	MP_BAK							: sMachPara;
END_VAR
VAR_IN_OUT
	sVisu : sMPHandler;
END_VAR
DisableMP();
j:=1;
FOR i:=1 TO 20 DO
	IF ExportDirectory[i].sFileName<>''
	THEN
		sVisu.FileListExport[j]:=ExportDirectory[i].sFileName;
		j:=j+1;
	ELSE
		sVisu.FileListExport[j]:='';
		j:=j+1;
	END_IF
END_FOR
j:=1;
FOR i:=1 TO 20 DO
	IF LocalDirectory[i].sFileName<>''
	THEN
		sVisu.FileListLocal[j]:=LocalDirectory[i].sFileName;
		j:=j+1;
	ELSE
		sVisu.FileListLocal[j]:='';
		j:=j+1;
	END_IF
END_FOR


(* --------------------------------------------------------------- *)
(* -----------------  sVisu interface ----------------------------- *)
(* --------------------------------------------------------------- *)



BtnImport(
	Enable			:= StepExport=0,
	Visible			:= FALSE,
	TextOn			:= 'Import',
	TextOff			:= 'Import',
	Button			:= sVisu.BtnImport
  );



BtnExport(
	Enable			:= StepExport=0,
	Visible			:= TRUE,
	TextOn			:= 'Export',
	TextOff			:= 'Export',
	Button			:= sVisu.BtnExport
  );

IF BtnExport.PressedFlag
THEN
StepExport:=1;

END_IF


CASE StepExport OF
(* Überprüfen ob Laufwerk vorh. ist *)
	0:	sVisu.MessageString:='';
	1:	FileNameSearchExport	:=	MP_ExportDrive;
			sVisu.MessageString:='';
			StepExport			:=	2(*2*);
	2:	FileListUpdateExport:=TRUE;
			StepExport			:=	3;
	3:	IF ExportFiles.bError OR (ExportFiles.bEOE AND ExportFiles.nFindFiles=0 AND NOT ExportFiles.bBusy)
			THEN
				sVisu.MessageString:='Exportlaufwerk wurde nichterkannt!';
				FileListUpdateExport:=FALSE;
				StepExport			:=	999;
			ELSIF ExportFiles.bEOE AND  ExportFiles.nFindFiles>0
			THEN
				FileListUpdateExport:=FALSE;
				StepExport			:=	4;
			END_IF
	4:	IF NOT ExportFiles.bBusy
			THEN
				StepExport			:=	10;
			END_IF
(* Typdaten Exportpfad prüfen / anlegen *)
	10:	FileNameSearchExport	:=	MP_ExportDrivePathTD;(* 4 *)
			sVisu.MessageString:='';
			StepExport			:=	11;
	11:	FileListUpdateExport:=TRUE;
			StepExport			:=	12;
	12:	IF ExportFiles.nFindFiles=0 AND (ExportFiles.bEOE OR ExportFiles.bError)
			THEN
				sVisu.MessageString:='Typdatenpfad wird angelegt! -> /_TD/';
				FileListUpdateExport:=FALSE;
				StepExport			:=	13;
			ELSIF ExportFiles.nFindFiles>0 AND (ExportFiles.bEOE OR ExportFiles.bError)
			THEN
				FileListUpdateExport:=FALSE;
				StepExport			:=	20;
			END_IF
	13:	CreateDirectory.sPathName:=MP_ExportDrivePathTD;
			CreateDirectory.bExecute:=FALSE;
			StepExport			:=	14;
	14:	CreateDirectory.bExecute:=TRUE;
			IF CreateDirectory.bBusy
			THEN
				StepExport			:=	15;
			END_IF
	15:	IF NOT CreateDirectory.bBusy AND NOT CreateDirectory.bError
			THEN
				StepExport			:=	20;

			ELSIF NOT CreateDirectory.bBusy AND CreateDirectory.bError
			THEN
				StepExport			:=	999;
				sVisu.MessageString:='Fehler bein erstellen des Typdatenpfades';
			END_IF


(* Maschinenparameter Exportpfad prüfen / anlegen *)
	20:	FileNameSearchExport	:=	MP_ExportDrivePathMP;
			sVisu.MessageString:='';
			StepExport			:=	21;
	21:	FileListUpdateExport:=TRUE;
			StepExport			:=	22;
	22:	IF ExportFiles.nFindFiles=0 AND (ExportFiles.bEOE OR ExportFiles.bError)
			THEN
				sVisu.MessageString:='Maschinenparameterpfad  wird angelegt! -> /_MP/';
				FileListUpdateExport:=FALSE;
				StepExport			:=	23;
			ELSIF ExportFiles.nFindFiles>0 AND (ExportFiles.bEOE OR ExportFiles.bError)
			THEN
				FileListUpdateExport:=FALSE;
				StepExport			:=	40;
			END_IF
	23:	CreateDirectory.sPathName:=MP_ExportDrivePathMP;
			CreateDirectory.bExecute:=FALSE;
			StepExport			:=	24;
	24:	CreateDirectory.bExecute:=TRUE;
			IF CreateDirectory.bBusy
			THEN
				StepExport			:=	25;
			END_IF
	25:	IF NOT CreateDirectory.bBusy AND NOT CreateDirectory.bError
			THEN
				StepExport			:=	40;

			ELSIF NOT CreateDirectory.bBusy AND CreateDirectory.bError
			THEN
				StepExport			:=	999;
				sVisu.MessageString:='Fehler bein erstellen des Maschinenparameterpfades';
			END_IF

	(* Typdaten kopieren *)
	40: sVisu.MessageString:='';
			StepExport			:=	41;
			FileNameSearchExport	:=	CONCAT(CONCAT(MP_ExportDrivePathTD,Backslash),MP_TDSearchString);
			FileNameSearchLocal		:=	CONCAT(MP_TDPathLocal,MP_TDSearchString);
	41: FileListUpdateExport:=TRUE;
			StepExport			:=	42;
	42: IF ExportFiles.bEOE OR ExportFiles.bError
			THEN
				FileListUpdateExport:=FALSE;
				StepExport			:=	43;
			END_IF
	43: FileListUpdateLocal:=TRUE;
			StepExport			:=	44;
	44: IF LocalFiles.nFindFiles=0 AND (LocalFiles.bEOE OR LocalFiles.bError)
			THEN
				sVisu.MessageString:='Es wurden keine Typdaten zum Exportieren gefunden!';
				FileListUpdateLocal:=FALSE;
				StepExport			:=	100;
			ELSIF LocalFiles.nFindFiles>0 AND (LocalFiles.bEOE OR LocalFiles.bError)
			THEN
				FileListUpdateLocal:=FALSE;
				NoOfTDFilesToCopy:=LocalFiles.nFindFiles;
				StepExport			:=	60;
			END_IF

	60:	AktFileToCopy		:=	1;
			StepExport			:=	61;

	61: (* Set Path *)
			TempStringSource					:=	CONCAT(MP_TDPathLocal,LocalDirectory[AktFileToCopy].sFileName);
			TempStringTarget					:=	CONCAT(CONCAT(MP_ExportDrivePathTD,Backslash),LocalDirectory[AktFileToCopy].sFileName);
			CopyFiles.srcFileName			:=	TempStringSource;
			CopyFiles.destFileName		:=	TempStringTarget;
			CopyFiles.bExecute				:=	FALSE;
			StepExport								:=	62;
			sVisu.MessageString:='Typdaten werden kopiert...';

	62: (* Start to Copy *)
			CopyFiles.bExecute				:=	TRUE;
			IF CopyFiles.bBusy
			THEN
				StepExport								:=	63;
			END_IF
	63: (* Copy Done *)
			CopyFiles.bExecute				:=	FALSE;
			IF NOT CopyFiles.bBusy AND NOT CopyFiles.bError
			THEN
				StepExport								:=	64;
			ELSIF NOT CopyFiles.bBusy AND CopyFiles.bError
			THEN
				StepExport								:=	999;
				sVisu.MessageString:='Fehler beim kopieren der Typdaten!';
			END_IF
	64: FileListUpdateExport:=TRUE;
			StepExport			:=	65;
	65:	(* Check last file To copy *)
			FileListUpdateExport:=FALSE;
			IF AktFileToCopy>=NoOfTDFilesToCopy
			THEN
				StepExport								:=	66;
			ELSE
				AktFileToCopy							:=	AktFileToCopy + 1;
				StepExport								:=	61;
			END_IF

	66:	(* All Files copied *)
			sVisu.MessageString:='Typdaten kopieren abgeschlossen!';
				StepExport								:=	100;

 100:	(* Maschinendaten sichern *)
			WriteXML.bExecute					:=	FALSE;
			StepExport								:=	101;
 101: WriteXML.bExecute					:=	TRUE;
			IF WriteXML.bBusy
			THEN
				WriteXML.bExecute					:=	FALSE;
				StepExport								:=	102;
			END_IF
 102: IF NOT WriteXML.bBusy AND NOT WriteXML.bError
			THEN
				WriteXML.bExecute					:=	FALSE;
				StepExport								:=	110;
			ELSIF NOT WriteXML.bBusy AND WriteXML.bError
			THEN
				sVisu.MessageString:='Fehler bein schreiben der XML-Datei für die Maschinenparameter....';
				WriteXML.bExecute					:=	FALSE;
				StepExport								:=	999;
			END_IF
 110:
			(* Set Path *)
			TempStringSource					:=	CONCAT(CONCAT(MP_ExportDrivePathMP, Backslash),MP_MPExportFilename);(*'\Hard Disk\_MP\MachPara.xml';*)
			TempStringTarget					:=	CONCAT(CONCAT(MP_ExportDrivePathMP, Backslash),MP_MPExportFilename);(*'\Hard Disk2\_MP\MachPara.xml';*)
			CopyFiles.srcFileName			:=	TempStringSource;
			CopyFiles.destFileName		:=	TempStringTarget;
			CopyFiles.bExecute				:=	FALSE;
			StepExport								:=	111;
			sVisu.MessageString:='Maschinenparameter werden kopiert...';

	111: (* Start to Copy *)
			CopyFiles.bExecute				:=	TRUE;
			IF CopyFiles.bBusy
			THEN
				StepExport								:=	112;
			END_IF
	112: (* Copy Done *)
			CopyFiles.bExecute				:=	FALSE;
			IF NOT CopyFiles.bBusy AND NOT CopyFiles.bError
			THEN
				sVisu.MessageString:='Maschinenparameter kopieren abgeschlossen!';
				StepExport								:=	999;
			ELSIF NOT CopyFiles.bBusy AND CopyFiles.bError
			THEN
				StepExport								:=	999;
				sVisu.MessageString:='Fehler beim kopieren der Maschinenparameter!';
			END_IF
 999:	Delay(IN:= FALSE, PT:= t#0s);
			StepExport			:=	1000;
1000: Delay(IN:= TRUE, PT:= t#1s);
			IF delay.Q
			THEN
				StepExport			:=	0;
			END_IF
END_CASE


ExportFiles(
	bExecute			:=sVisu.FileListUpdate OR FileListUpdateExport,
	sNetId				:= '',
	sPathName			:= FileNameSearchExport,
	pFindList			:= ADR(ExportDirectory),
	cbFindList		:= SIZEOF(ExportDirectory) ,
	tTimeout			:= t#10s );

LocalFiles(
	bExecute			:=sVisu.FileListUpdate OR FileListUpdateLocal,
	sNetId				:= '',
	sPathName			:= FileNameSearchLocal,
	pFindList			:= ADR(LocalDirectory),
	cbFindList		:= SIZEOF(LocalDirectory) ,
	tTimeout			:= t#1s );

CopyFiles(
	srcNetId:= '',
	destNetId:= '',
	tAdsSTATE_TIMEOUT:= t#1s);


WriteXML(
	sNetId				:= '',
	nMode					:= XMLSRV_ADDMISSING,
 	sSymName				:='.MP',
	sFilePath			:= CONCAT(CONCAT(MP_ExportDrivePathMP, Backslash),MP_MPExportFilename),
	sXPath				:= '/dataentry/MP',
	tTimeout			:= t#10s );


sVisu.FileListUpdate:=FALSE;

CreateDirectory(
	sNetId:= '' );


ReadXML(
	sNetId:= '',
	nMode:= XMLSRV_ADDMISSING,
	sSymName:= '.MP',
	sFilePath:= '\Hard Disk\_MP\MachPara.xml',
	sXPath:= '/dataentry/MP'
);


IF MEMCMP(ADR(MP),ADR(MP_BAK),SIZEOF(MP_BAK))<>0
THEN
	Visu.SavePersistentData:=TRUE;
	MP_BAK:=MP;
END_IF
END_PROGRAM
ACTION DisableMP:
(* Sperre der Typdateneingabe *)
gDisableMP := FALSE;
IF 	CurrentUserLevel <6  OR
	ModeSelect.Mode > MODE_MANUAL THEN
	gDisableMP := TRUE;
END_IF
END_ACTION

(* POU System/HelpFunctions/FB_FileCopy, ST *)
FUNCTION_BLOCK FB_FileCopy
VAR_INPUT
	srcNetId				: T_AmsNetId;	(* TwinCAT network address of the source file *)
	srcFileName				: T_MaxString;	(* source file path and name *)
	destNetId				: T_AmsNetId;	(* TwinCAT network address of the destination file *)
	destFileName			: T_MaxString;  	(* destination file path and name *)
	bExecute				: BOOL;		(* rising edge starts fb execution *)
	tAdsSTATE_TIMEOUT	: TIME;		(* ads STATE_TIMEOUT *)
END_VAR
VAR_OUTPUT
	bBusy		  		:BOOL;
	bError				:BOOL;
	nErrId				:UDINT;
END_VAR
VAR
	fbFileOpen			:FB_FileOpen;
	fbFileClose			:FB_FileClose;
	fbFileRead			:FB_FileRead;
	fbFileWrite			:FB_FileWrite;

	hSrcFile				:UINT	:= 0;(* file handle of the source file *)
	hDestFile			:UINT	:= 0;(* file handle of the destination file *)

	Step				:DWORD;
	RisingEdge			:R_TRIG;

	buffRead			:ARRAY[1..100000] OF BYTE;(* buffer *)
	cbReadLength		:UDINT:=0;
END_VAR
RisingEdge(CLK:=bExecute);
IF RisingEdge.Q THEN
	IF 	NOT bBusy THEN
		bBusy := TRUE;
		bError:= FALSE;
		nErrId:=0;
		Step := 1;
		cbReadLength:=0;
		hSrcFile:=0;
		hDestFile:=0;
	END_IF
END_IF


CASE Step OF
	0:(* do nothing *)
	;

	1:(* open source file *)
	fbFileOpen(  bExecute := FALSE  );
	fbFileOpen(	sNetId := srcNetId,
		sPathName := srcFileName,
		nMode := FOPEN_MODEREAD OR FOPEN_MODETEXT ,
		ePath := PATH_GENERIC,
		tTimeout := tAdsSTATE_TIMEOUT,
		bExecute := TRUE );
		Step := Step + 1;

	2:
	fbFileOpen( bExecute := FALSE );
	IF ( NOT fbFileOpen.bBusy ) THEN
		IF ( fbFileOpen.bError ) THEN
			nErrId := fbFileOpen.nErrId;
			bError := TRUE;
			Step := 50;
		ELSE
			hSrcFile := fbFileOpen.hFile;
			Step := Step + 1;
		END_IF
	END_IF

	3:(* open destination file *)
	fbFileOpen(  bExecute := FALSE  );
	fbFileOpen( 	sNetId := destNetId,
			sPathName := destFileName,
			nMode := FOPEN_MODEWRITE OR FOPEN_MODETEXT ,
			ePath := PATH_GENERIC,
			tTimeout := tAdsSTATE_TIMEOUT,
			bExecute := TRUE );
	Step := Step+1;

	4:
	fbFileOpen(  bExecute := FALSE  );
	IF ( NOT fbFileOpen.bBusy ) THEN
		IF ( fbFileOpen.bError ) THEN
			nErrId := fbFileOpen.nErrId;
			bError := TRUE;
			Step := 50;
		ELSE
			hDestFile := fbFileOpen.hFile;
			Step := Step + 1;
		END_IF
	END_IF

	5:(*read data from source file*)
	cbReadLength := 0;
	fbFileRead( bExecute:= FALSE );
	fbFileRead( 	sNetId:=SrcNetId,
			hFile:=hSrcFile,
			pReadBuff:= ADR(buffRead),
			cbReadLen:= SIZEOF(buffRead),
			bExecute:=TRUE,
			tTimeout:=tAdsSTATE_TIMEOUT );
	Step := Step + 1;

	6:
	fbFileRead( bExecute:= FALSE );
	IF ( NOT fbFileRead.bBusy ) THEN
		IF ( fbFileRead.bError ) THEN
			nErrId := fbFileRead.nErrId;
			bError := TRUE;
			Step := 50;
		ELSE
			cbReadLength := fbFileRead.cbRead;
			Step := Step + 1;
		END_IF
	END_IF

	7:(*write data to destination file*)
	fbFileWrite( bExecute := FALSE );
	fbFileWrite(	sNetId:=DestNetId,
			hFile:=hDestFile,
			pWriteBuff:= ADR(buffRead),
			cbWriteLen:= cbReadLength,
			bExecute:=TRUE,
			tTimeout:=tAdsSTATE_TIMEOUT );
	Step := Step + 1;

	8:
	fbFileWrite( bExecute := FALSE );
	IF ( NOT fbFileWrite.bBusy ) THEN
		IF ( fbFileWrite.bError ) THEN
			nErrId := fbFileWrite.nErrId;
			bError := TRUE;
			Step := 50;
		ELSE
			IF fbFileRead.bEOF THEN (*Check if the EOF flag ist set *)
				Step := 50;(*cleanup: close the destination and source files *)
			ELSE
				Step := 5; (* repeat reading *)
			END_IF
		END_IF
	END_IF

	30:(* close the destination file *)
	fbFileClose( bExecute := FALSE );
	fbFileClose( 	sNetId:=destNetId,
			hFile:=hDestFile,
			bExecute:=TRUE,
			tTimeout:=tAdsSTATE_TIMEOUT );
	Step := Step + 1;

	31:
	fbFileClose( bExecute := FALSE );
	IF ( NOT fbFileClose.bBusy ) THEN
		IF ( fbFileClose.bError ) THEN
			nErrId := fbFileClose.nErrId;
			bError := TRUE;
		END_IF
		Step := 50;
		hDestFile := 0;
	END_IF

	40: (* close source file *)
	fbFileClose( bExecute := FALSE );
	fbFileClose( 	sNetId:=srcNetId,
			hFile:=hSrcFile,
			bExecute:=TRUE,
			tTimeout:=tAdsSTATE_TIMEOUT );
	Step := Step + 1;

	41:
	fbFileClose( bExecute := FALSE );
	IF ( NOT fbFileClose.bBusy ) THEN
		IF ( fbFileClose.bError ) THEN
			nErrId := fbFileClose.nErrId;
			bError := TRUE;
		END_IF
		Step := 50;
		hSrcFile := 0;
	END_IF

	50: (*error or ready => cleanup*)
	IF ( hDestFile <> 0 ) THEN
		Step := 30; (* close the destination file*)
	ELSIF (hSrcFile <> 0 ) THEN
		Step := 40; (* close the source file *)
	ELSE
		Step := 0;	(* ready *)
		bBusy := FALSE;
	END_IF

END_CASE
END_FUNCTION_BLOCK

(* POU System/MP_ShiftHandler/MP_ShiftHandler, ST *)
PROGRAM MP_ShiftHandler
VAR
	TodNow				: TOD;

	TempStartTOD 		: TOD;
	TempEndTOD 			: TOD;

	TempNightShift		: BOOL;

	TimeDayBegins		: TOD := TOD#00:00;
	TimeDayEnds			: TOD := TOD#23:59:59.999;

	NumberofShifts		: DINT;
	Idx					: DINT;

	NoShiftActive		: sMP_ShiftData;
	OneShiftIsActive	: BOOL;

END_VAR
NoShiftActive.ShiftIndex:=999;
NoShiftActive.ShiftName:='keine Schicht Activ';


NumberofShifts:=SIZEOF(MP.ShiftData.Shift)/SIZEOF(mp.ShiftData.ActiveShift);

TodNow:=DT_TO_TOD(SYSTEMTIME_TO_DT(gVarSystemtime));
TodNow:=	DINT_TO_TOD(TOD_TO_DINT(TodNow)	+	WORD_TO_DINT(gVarSystemtime.wMilliseconds));


OneShiftIsActive:=FALSE;

FOR Idx:=1 TO NumberofShifts DO


	MP.ShiftData.Shift[Idx].TimeStart.wYear:=gVarSystemtime.wYear;
	MP.ShiftData.Shift[Idx].TimeStart.wMonth:=gVarSystemtime.wMonth;
	MP.ShiftData.Shift[Idx].TimeStart.wDay:=gVarSystemtime.wDay;
	MP.ShiftData.Shift[Idx].TimeStart.wDayOfWeek:=gVarSystemtime.wDayOfWeek;
	MP.ShiftData.Shift[Idx].TimeStart.wSecond:=0;
	MP.ShiftData.Shift[Idx].TimeStart.wMilliseconds:=0;


	MP.ShiftData.Shift[Idx].TimeEnd.wYear:=gVarSystemtime.wYear;
	MP.ShiftData.Shift[Idx].TimeEnd.wMonth:=gVarSystemtime.wMonth;
	MP.ShiftData.Shift[Idx].TimeEnd.wDay:=gVarSystemtime.wDay;
	MP.ShiftData.Shift[Idx].TimeEnd.wDayOfWeek:=gVarSystemtime.wDayOfWeek;
	MP.ShiftData.Shift[Idx].TimeEnd.wSecond:=59;
	MP.ShiftData.Shift[Idx].TimeEnd.wMilliseconds:=0;


	TempStartTOD:=DT_TO_TOD(SYSTEMTIME_TO_DT(MP.ShiftData.Shift[Idx].TimeStart));

	TempStartTOD:=	DINT_TO_TOD(TOD_TO_DINT(TempStartTOD)	+	WORD_TO_DINT(MP.ShiftData.Shift[Idx].TimeStart.wMilliseconds));

	TempEndTOD:=DT_TO_TOD(SYSTEMTIME_TO_DT(MP.ShiftData.Shift[Idx].TimeEnd));

	MP.ShiftData.Shift[Idx].TimeEnd.wMilliseconds:=999;
	TempEndTOD:=	DINT_TO_TOD(TOD_TO_DINT(TempEndTOD)	+	WORD_TO_DINT(MP.ShiftData.Shift[Idx].TimeEnd.wMilliseconds));


	TempNightShift:=TOD_TO_DINT(TempStartTOD)>TOD_TO_DINT(TempEndTOD);

	IF 	NOT TempNightShift THEN
		MP.ShiftData.Shift[Idx].ShiftActive:=	(TodNow >= TempStartTOD)	AND (TodNow <= TempEndTOD);
	ELSE
		MP.ShiftData.Shift[Idx].ShiftActive:=	(TodNow >= TempStartTOD) AND
											(TodNow <= TimeDayEnds) OR (TodNow >= TimeDayBegins) AND
											(TodNow <= TempEndTOD);
	END_IF

	IF 	NOT OneShiftIsActive THEN
		OneShiftIsActive:=MP.ShiftData.Shift[Idx].ShiftActive;
		MP.ShiftData.ActiveShift:=MP.ShiftData.Shift[Idx];
	END_IF

END_FOR

IF 	NOT OneShiftIsActive THEN
	MP.ShiftData.ActiveShift:=NoShiftActive;
END_IF
END_PROGRAM

(* POU Stations/ST_00/ST00_FBs/_CallFBs, ST *)
PROGRAM _CallFBs


VAR



END_VAR
ST00_CallFBs();
ST03_CallFBs();

ST08_CallFBs();
END_PROGRAM

(* POU Stations/ST_00/ST00_FBs/ST00_CallFBs, ST *)
PROGRAM ST00_CallFBs
(*   Author:           *)


VAR



END_VAR
(* ----------------------------------------------------------------------------------------- *)
(* 																				Eingänge  																				 *)
(* ----------------------------------------------------------------------------------------- *)


(* Call ST00_40_F1 Vorsicherungen Leistung iO (DigIn) *)
ST00_40_F1(	sVisu:=Visu.ST00_40_F1,
			Reset:=gResetAll,
			CheckSignalHigh:=TRUE,
);

(* Call ST03_210_S1 Not-Aus 1 Anlage ausgelöst (DigIn) *)
ST03_210_S1(	sVisu:=Visu.ST03_210_S1,
				Reset:=gResetAll,
				CheckSignalLow:=TRUE,
);
(* Call ST08_210_S2 Not-Aus 2 Anlage ausgelöst (DigIn) *)
ST08_210_S2(	sVisu:=Visu.ST08_210_S2,
				Reset:=gResetAll,
				CheckSignalLow:=FALSE,
				CheckSignalHigh:=TRUE,
);

(* Call ST00_X4_16  Not-Halt 2 Tampondrucker  (DigIn) *)
ST00_X4_16(	sVisu:=Visu.ST00_X4_16,
			Reset:=gResetAll,
			CheckSignalLow:=TRUE,
);

(* Call ST00_200_A1_A1 Not-Aus iO (DigIn) *)
ST00_200_A1_A1(	sVisu:=Visu.ST00_200_A1_A1,
				Reset:=gResetAll,
				CheckSignalHigh:=TRUE,
);

(* Call ST00_220_S1 Schutztüre 1 geöffnet (DigIn) *)
ST00_220_S1(sVisu:=Visu.ST00_220_S1,
			Reset:=gResetAll,
			CheckSignalLow:=TRUE,
);

(* Call ST00_220_S2 Schutztüre 1 geöffnet (DigIn) *)
ST00_220_S2(sVisu:=Visu.ST00_220_S2,
			Reset:=gResetAll,
			CheckSignalLow:=TRUE,
);

(* Call ST00_230_S2_E1 Schutztüre 1 geschlossen (DigIn) *)
ST00_230_S2_E1(sVisu:=Visu.ST00_230_S2_E1,
			Reset:=gResetAll,
			(* CheckSignalHigh:=TRUE,*) (* @@@ *)
);

(* Call ST00_240_S1 Schutztüre 9 geschlossen (DigIn) *)
ST00_240_S1(sVisu:=Visu.ST00_240_S1,
			Reset:=gResetAll,
);

(* Call ST00_226_S1 Hubtüre 1 Schleuse Einlauf STN 8 geschlossen (DigIn) *)
ST00_226_S1(sVisu:=Visu.ST00_226_S1,
			Reset:=gResetAll,
);
(* Call ST00_226_S2 Hubtüre 2 Schleuse Einlauf STN 8 geschlossen (DigIn) *)
ST00_226_S2(sVisu:=Visu.ST00_226_S2,
			Reset:=gResetAll,
);
(* Call ST00_227_S1 Hubtüre 3 Schleuse Auslauf STN 8 geschlossen (DigIn) *)
ST00_227_S1(sVisu:=Visu.ST00_227_S1,
			Reset:=gResetAll,
);
(* Call ST00_227_S2 Hubtüre 4 Schleuse Auslauf STN 8 geschlossen (DigIn) *)
ST00_227_S2(sVisu:=Visu.ST00_227_S2,
			Reset:=gResetAll,
);
(* Call ST00_229_S1 Schutztüre Einlauf Tray STN 8 geschlossen (DigIn) *)
ST00_229_S1(sVisu:=Visu.ST00_229_S1,
			Reset:=gResetAll,
);
(* Call ST00_230_S1 Schutztüre Auslauf Tray STN 8 geschlossen (DigIn) *)
ST00_230_S1(sVisu:=Visu.ST00_230_S1,
			Reset:=gResetAll,
);
(* Call ST00_231_S1 Schutztüre Panel / Rutsche STN 8 geschlossen (DigIn) *)
ST00_231_S1(sVisu:=Visu.ST00_231_S1,
			Reset:=gResetAll,
);
(* Call ST00_232_S1 Schutztüre 8 Auslauf Tray STN 8 geschlossen (DigIn) *)
ST00_232_S1(sVisu:=Visu.ST00_232_S1,
			Reset:=gResetAll,
);
(* Call ST00_170Motorschutz Motorschutz in Ordnung (DigIn) *)
ST00_170_Motorschutz( sVisu:=Visu.ST00_170_Motorschutz,
						Reset:=gResetAll,
						CheckSignalHigh:=TRUE,
);

(* Call ST00_Thermokont Thermokontakt in Ordnung (DigIn) *)
ST00_170_Thermokont(	sVisu:=Visu.ST00_170_Thermokont,
						Reset:=gResetAll,
						CheckSignalHigh:=TRUE,
);


(* Call ST00_228_S1 Pallettierer in Position (DigIn) *)
ST00_228_S1(sVisu:=Visu.ST00_228_S1,
			Reset:=gResetAll,
);

(* Call ST00_71_X1_3 Schnittstelle Bedrucken Tinte JSK auf Übergabeposition (DigIn) *)
ST00_71_X1_3(sVisu:=Visu.ST00_71_X1_3,
			Reset:=gResetAll,
);

(* Call ST00_71_X1_4 Schnittstelle Bedrucken Tinte Druckstation betriebsbereit (DigIn) *)
ST00_71_X1_4(sVisu:=Visu.ST00_71_X1_4,
			Reset:=gResetAll,
);

(* Call ST00_72_X1_3 Schnittstelle Tampondrucker Teil in Abholposition (DigIn) *)(*Band Entnahmeposition 1*)
ST00_72_X1_3(sVisu:=Visu.ST00_72_X1_3,
			Reset:=gResetAll,
);

(* Call ST00_72_X1_8 Schnittstelle Tampondrucker Druck abgeschlossen (DigIn) *)
ST00_72_X1_8(sVisu:=Visu.ST00_72_X1_8,
			Reset:=gResetAll,
);

(* Call ST00_292_S1_STOP Bedienstelle Produktion Stop (DigIn) *)
ST00_292_S1_STOP(	sVisu:=Visu.ST00_292_S1_STOP,
					Reset:=gResetAll,
);
(* Call ST00_292_S2_START Bedienstelle Produktion Start (DigIn) *)
ST00_292_S2_START(	sVisu:=Visu.ST00_292_S2_START,
					Reset:=gResetAll,
);

(* Call ST00_292_S3_RESET Bedienstelle Produktion Start (DigIn) *)
ST00_292_S3_RESET(	sVisu:=Visu.ST00_292_S3_RESET,
					Reset:=gResetAll,
);
(* Call ST00_350_B20_0 Druckschalter Wartungseinheit Hauptluft min.6 bar (DigIn) *)
ST00_350_B20_0(	sVisu:=Visu.ST00_350_B20_0,
				Reset:=gResetAll,
				CheckSignalHigh:=TRUE,
);

(* Call 	ST00_245_V1			Verriegelung Schutztüren-Leuchte (DigOutIn) *)
ST00_245_V1(	sVisu:=Visu.ST00_245_V1,
					Reset:=gResetAll,
);

(* Call 	ST00_245_V2_START	Bedienstelle Start-Leuchte (DigOutIn) *)
ST00_245_V2_START(	sVisu:=Visu.ST00_245_V2_START,
					Reset:=gResetAll,
);

(* Call 	ST00_245_V3_RESET	Bedienstelle Reset-Schutztüren-Leuchte (DigOutIn) *)
ST00_245_V3_RESET(	sVisu:=Visu.ST00_245_V3_RESET,
					Reset:=gResetAll,
);

(* Call 	ST00_245_S1_STOP 	Bedienstelle Produktion Stop (DigIn) *)
ST00_245_S1_STOP(	sVisu:=Visu.ST00_245_S1_STOP,
					Reset:=gResetAll,
);

(* Call 	ST00_245_S2_START	Bedienstelle Produktion Start (DigIn) *)
ST00_245_S2_START(	sVisu:=Visu.ST00_245_S2_START,
					Reset:=gResetAll,
);

(* Call 	ST00_245_S3_RESET	Bedienstelle Produktion Reset (DigIn) *)
ST00_245_S3_RESET(	sVisu:=Visu.ST00_245_S3_RESET,
					Reset:=gResetAll,
);

(* ----------------------------------------------------------------------------------------- *)
(* 																				Ausgänge																					 *)
(* ----------------------------------------------------------------------------------------- *)

(* Call ST00_31_K1 Beleuchtung Anlage (DigOutIn) *)
ST00_31_K1(	sVisu:=Visu.ST00_31_K1,
			Reset:=gResetAll,
);

(* Call ST00_350_H1 Signalsäule RD Maschine Alarm/Störung (DigOutIn) *)
ST00_350_H1(sVisu:=Visu.ST00_350_H1,
			Reset:=gResetAll,
);

(* Call ST00_350_H2 Signalsäule YE Bedienereingriff erforderlich (DigOutIn) *)
ST00_350_H2(sVisu:=Visu.ST00_350_H2,
			Reset:=gResetAll,
);

(* Call ST00_350_H3 Signalsäule GN Maschine Automatik (DigOutIn) *) 
ST00_350_H3(sVisu:=Visu.ST00_350_H3,
			Reset:=gResetAll,
);

(* Call ST00_200_A1_E4 Quittierung Not-Aus (DigOutIn) *)
ST00_200_A1_E4(	sVisu:=Visu.ST00_200_A1_E4,
				Reset:=gResetAll,
);

(* Call ST00_220_S1_S31 Verriegelung Schutztüren (DigOutIn) *)
ST00_220_S1_S31                (sVisu:=Visu.ST00_220_S1_S31,
			Reset:=gResetAll,
);

(* Call ST00_292_H2_START Bedienstelle Start-Leuchte (DigOutIn) *)
ST00_292_H2_START(	sVisu:=Visu.ST00_292_H2_START,
					Reset:=gResetAll,
);

(* Call ST00_292_H3_RESET Bedienstelle Reset-Leuchte (DigOutIn) *)
ST00_292_H3_RESET(	sVisu:=Visu.ST00_292_H3_RESET,
					Reset:=gResetAll,
);

(* Call ST00_71_K2 Schnittstelle Bedrucken Tinte Abholposition frei (DigOutIn) *)
ST00_71_K2(	sVisu:=Visu.ST00_71_K2,
			Reset:=gResetAll,
);

(*  Call ST00_73_K3 Schnittstelle Förderband frei für Spritzmaschine*)
ST00_73_K3(	sVisu:=Visu.ST00_73_K3,
			Reset:=gResetAll,
);
(* Call ST00_73_K4   Schnittstelle Freigabe von Spritzmaschine (nur für Anlagen ohne Rundtisch) (DigIn) *)
ST00_73_K4(	sVisu:=Visu.ST00_73_K4,
			Reset:=gResetAll,
			CheckSignalHigh:=FALSE,
);
(* Call ST00_74_Y2_4 Vereinzeler Bandstrecke (Valve) *)
Analyze(	InputExp:=  TRUE,
			DoAnalyze:= TRUE );
ST00_74_Y2_4.strAnlayse:=Analyze.OutString;
ST00_74_Y2_4(	Enable  :=  Analyze.ExpResult,
				sVisu:=Visu.ST00_74_Y2_4,
				Reset:=gResetAll,
);
ST00_74_B7_2(ValveObject:= ADR(ST00_74_Y2_4));(*Vereinzeler GST1 DS*)
ST00_74_B7_3(ValveObject:= ADR(ST00_74_Y2_4));(*Vereinzeler GST2 PS*)


(* Call ST00_74_Y2_5 Vereinzeler Bandstrecke (Valve) *)
Analyze(	InputExp:=  TRUE,
			DoAnalyze:= TRUE );
ST00_74_Y2_5.strAnlayse:=Analyze.OutString;
ST00_74_Y2_5(	Enable  :=  Analyze.ExpResult,
				sVisu:=Visu.ST00_74_Y2_5,
				Reset:=gResetAll,
);
ST00_74_B7_4(ValveObject:= ADR(ST00_74_Y2_5));(*Vereinzeler AST1 DS*)
ST00_74_B7_6(ValveObject:= ADR(ST00_74_Y2_5));(*Vereinzeler GST1 DS*)
ST00_74_B7_5(ValveObject:= ADR(ST00_74_Y2_5));(*Vereinzeler AST2 PS*)
ST00_74_B7_7(ValveObject:= ADR(ST00_74_Y2_5));(*Vereinzeler GST2 PS*)
END_PROGRAM

(* POU Stations/ST_03_Ruestsaetze/ST_03_FBs/ST03_CallFBs, ST *)
PROGRAM ST03_CallFBs
VAR

	ST03_463_B70_3_4_pos	:INT;

END_VAR
(*Bei NOX4 darf der Override nicht größer 5 sein*)
IF gTypeCode=5631 AND MP.ST02.Override_Band>5 THEN
	MP.ST02.Override_Band:=5;
END_IF

(*Call ST03_51_M1 Förderbandmotor*)
ST03_51_M1			(sVisu:=Visu.ST03_51_M1,
						Override:= MP.ST02.Override_Band,
						Offset:=0,								(* in mm oder Grad am Abtrieb*)
						Reset:=gResetAll,
						NotausOK := TRUE);
(* ----------------------------------------------------------------------------------------- *)
(* 																	Roboter																									 *)
(* ----------------------------------------------------------------------------------------- *)

Robot01.sToolSettings.NameCoilA:='120_A1_A12';
Robot01.sToolSettings.NameCoilB:='xxxx';
Robot01.sToolSettings.NameInitSensor:='400_B12_4';
Robot01.sToolSettings.NameWorkSensor:='400_B12_5';
Robot01.sToolSettings.NameBtnToolOn:='Greifer Öffnen';
Robot01.sToolSettings.NameBtnToolOff:='Greifer Schliessen';

Analyze         (InputExp:=  ST03_Init_Lockings.InputExp_Robot01,
                 DoAnalyze:= TRUE );
Robot01(sVisu			:=visu.Robot01,
        Reset			:=gResetAll,
				Enable		:=TRUE,
				Acc				:=100,
				Vel				:=100,
				PosOffset :=gRobotOffset,
				strAnlayse:=Analyze.OutString,
				Override	:=MP.ST00.Override,
				CollisionActivated := MP.ST03.RoboterColisionActivated,
				Tool2Unit_AST :=ST03_400_B12_7.BitInToCheck);

(* ----------------------------------------------------------------------------------------- *)
(* 																	Eingänge																								 *)
(* ----------------------------------------------------------------------------------------- *)

(* Call ST03_125_F1 Absicherung Roboter iO (DigIn) *)
ST03_125_F1                    (sVisu:=Visu.ST03_125_F1,
                                Reset:=gResetAll,
																CheckSignalHigh:=TRUE,
);

(* Init ST03_A5 Bandantrieb Förderbandmotor Oriental (nur 3621) Ein (DigOutIn)*)
ST03_A5                  (sVisu:=Visu.ST03_A5,
                                Reset:=gResetAll,
);

(* Init ST03_601V1_A1 Förderband Prüfteile  (DigOutIn)*)
ST03_601V1_A1                  (sVisu:=Visu.ST03_601V1_A1,
                                Reset:=gResetAll,
);

(* Init ST03_V2 Störung Motor Förderband Oriental (DigIn) *)
ST03_V2                (sVisu:=Visu.ST03_V2,
                                Reset:=gResetAll,
);

(* Call ST03_120_A1:A14 Roboter Schwenkmodul ist ein (DigIn) *)
ST03_120_A1_A14                (sVisu:=Visu.ST03_120_A1_A14,
                                Reset:=gResetAll,
);

(* Call ST03_400_B12_6 Schwenkmodul AST (Roboterkopf) (DigIn) *)
ST03_400_B12_6                (sVisu:=Visu.ST03_400_B12_6,
                                Reset:=gResetAll,
);
(* Call ST03_400_B12_7 Schwenkmodul GST (Roboterkopf) (DigIn) *)
ST03_400_B12_7                (sVisu:=Visu.ST03_400_B12_7,
                                Reset:=gResetAll,
);
(* Call ST03_400_B54_7 Tray Testteile in Position (DigIn) *)
ST03_400_B54_7                (sVisu:=Visu.ST03_400_B54_7,
                                Reset:=gResetAll,
);
(* Call ST03_8_75_B13_5 voll/belegt keine Prüfmittel mehr (DigIn) *)
ST03_8_75_B13_5                (sVisu:=Visu.ST03_8_75_B13_5,
                                Reset:=gResetAll,
);
(* Call ST03_8_75_B13_6 belegt mit 6 Prüfmittel (DigIn) *)
ST03_8_75_B13_6                (sVisu:=Visu.ST03_8_75_B13_6,
                                Reset:=gResetAll,
);

(* Call ST03_BG3_X53_0 LED Taster Start Dummyprüfung Band (DigOutIn) *)
ST03_BG3_X53_0                  (sVisu:=Visu.ST03_BG3_X53_0,
                                Reset:=gResetAll,
);

(* Call ST03_65_Q1 Kühltunnel (Lüfter) (DigOutIn) *)
ST03_65_Q1                  (sVisu:=Visu.ST03_65_Q1,
                                Reset:=gResetAll,
);
(* Call ST03_65_F1 Sicherung Kühltunnel (Lüfter) *)
ST03_65_F1                (sVisu:=Visu.ST03_65_F1,
                                Reset:=gResetAll,
);

IF 	MP.ST03.SGM_3621 THEN
	(* Call ST03_Y01 Einschaltventil Hauptluft Tintenstrahldrucker (Valve) *)
	Analyze         (InputExp:=  TRUE,
	                 DoAnalyze:= TRUE );
	ST03_Y01.strAnlayse:=Analyze.OutString;
	ST03_Y01               (Enable  :=  Analyze.ExpResult,
	                                sVisu:=Visu.ST03_Y01,
	                                Reset:=gResetAll,
	);
END_IF

CASE  gTypeCode OF

4872:	call_154polRP();

4871:	call_154pol();

360, 379, 4992,489,322:	call_74_91_35_168_160pol();

522:		call_206pol();

550:		call_92pol();

564:		call_124pol();

569:		call_46pol();

5632,5633:	call_NOX5_6pol();

5631:	call_NOX4pol();

5731:	call_88pol();

575,5753,5754,5755:	call_7pol();

5732:	call_88polAMG();

5771:	call_120pol();

5772:	call_21pol();

580:	call_191pol();

5831:	call_72pol();

5832:	call_48pol();

5841, 4993:	call_268pol_102pol_neu();

5842:	call_268polRP();

598:	call_33pol();

END_CASE
END_PROGRAM
ACTION call_120pol:
(* Call ST03_531_B69_0 IZuführung  frei zum Ablegen ISK SP Maschine (DigIn) *)
ST03_531_B69_0(sVisu:=Visu.ST03_531_B69_0,
                                Reset:=gResetAll,
);
(* Call ST03_532_Y70_1  Zuführung Vereinzler AST/GST  (Valve) *)
Analyze(InputExp:=  TRUE, DoAnalyze:= TRUE );
ST03_532_Y70_1.strAnlayse:=Analyze.OutString;
ST03_532_Y70_1(Enable  :=  Analyze.ExpResult,
                                sVisu:=Visu.ST03_532_Y70_1,
                                Reset:=gResetAll,
);
ST03_531_B69_1(ValveObject:= ADR(ST03_532_Y70_1));(*  Zuführung Vereinzler eingefahren GST*)
ST03_531_B69_2(ValveObject:= ADR(ST03_532_Y70_1));(*  Zuführung Vereinzler ausgefahren AST*)

(* Call ST03_532_Y70_2  Züführung Stopper AST/GST  (Valve) *)
Analyze(InputExp:=  TRUE, DoAnalyze:= TRUE );
ST03_532_Y70_2.strAnlayse:=Analyze.OutString;
ST03_532_Y70_2(Enable  :=  Analyze.ExpResult,
                                sVisu:=Visu.ST03_532_Y70_2,
                                Reset:=gResetAll,
);
ST03_531_B69_3(ValveObject:= ADR(ST03_532_Y70_2));(* Zuführung Stopper  eingefahren  AST*)
ST03_531_B69_4(ValveObject:= ADR(ST03_532_Y70_2));(* Zuführung Stopper  ausgefahren GST*)


(* Call ST03_531_B69_6 SK anwesend am Stoper (DigIn) *)
ST03_531_B69_6(sVisu:=Visu.ST03_531_B69_6,
                                Reset:=gResetAll,
);
(* Call ST03_531_B69_7 ISK rechts Lageerkennung (DigIn) *)
ST03_531_B69_7(sVisu:=Visu.ST03_531_B69_7,
                                Reset:=gResetAll,
);
(* Call ST03_532_B70_0  ISK links Lageerkennung (DigIn) *)
ST03_532_B70_0(sVisu:=Visu.ST03_532_B70_0,
                                Reset:=gResetAll,
);
END_ACTION
ACTION call_124pol:
(* Call ST03_453_Y70_5 Förderband  Zuführung Vereinzler AST/GST  (Valve) *)
Analyze(InputExp:=  TRUE, DoAnalyze:= TRUE );
ST03_453_Y70_5.strAnlayse:=Analyze.OutString;
ST03_453_Y70_5(Enable  :=  Analyze.ExpResult,
                                sVisu:=Visu.ST03_453_Y70_5,
                                Reset:=gResetAll,
);
ST03_451_B69_0(ValveObject:= ADR(ST03_453_Y70_5));(*Förderband Zuführung Vereinzler   AST*)
ST03_451_B69_1(ValveObject:= ADR(ST03_453_Y70_5));(*Förderband Zuführung Vereinzler   GST*)

(* Call ST03_453_Y70_6 Förderband  Zuführung Stopper AST/GST  (Valve) *)
Analyze(InputExp:=  TRUE, DoAnalyze:= TRUE );
ST03_453_Y70_6.strAnlayse:=Analyze.OutString;
ST03_453_Y70_6(Enable  :=  Analyze.ExpResult,
                                sVisu:=Visu.ST03_453_Y70_6,
                                Reset:=gResetAll,
);
ST03_451_B69_2(ValveObject:= ADR(ST03_453_Y70_6));(*Förderband Zuführung Stopper   AST*)
ST03_451_B69_3(ValveObject:= ADR(ST03_453_Y70_6));(*Förderband Zuführung Stopper   GST*)

(* Call ST03_451_B69_4 Zuführung  frei zum Ablegen ISK SP Maschine Pos.1  (DigIn) *)
ST03_451_B69_4(sVisu:=Visu.ST03_451_B69_4,
                                Reset:=gResetAll,
);
(* Call ST03_451_B69_7 Zuführung  ISK anwesend am Stopper (DigIn) *)
ST03_451_B69_7(sVisu:=Visu.ST03_451_B69_7,
                                Reset:=gResetAll,
);
(* Call ST03_453_B70_4  ISK auf Übergabeposition zu Roboter  (DigIn) *)
ST03_453_B70_4(sVisu:=Visu.ST03_453_B70_4,
                                Reset:=gResetAll,
);
(* Call ST03_452_B70_1 Zuführung  ISK Lageerkennung links (DigIn) *)
ST03_452_B70_1(sVisu:=Visu.ST03_452_B70_1,
                                Reset:=gResetAll,
);
(* Call ST03_452_B70_2 Zuführung  ISK Lageerkennung links (DigIn) *)
ST03_452_B70_2(sVisu:=Visu.ST03_452_B70_2,
                                Reset:=gResetAll,
);
END_ACTION
ACTION call_154pol:
(* Call ST03_426_Y68_5 Förderband  Zuführung Vereinzler AST/GST  (Valve) *)
Analyze(InputExp:=  TRUE, DoAnalyze:= TRUE );
ST03_426_Y68_5.strAnlayse:=Analyze.OutString;
ST03_426_Y68_5(Enable  :=  Analyze.ExpResult,
                                sVisu:=Visu.ST03_426_Y68_5,
                                Reset:=gResetAll,
);
ST03_425_B67_0(ValveObject:= ADR(ST03_426_Y68_5));(*Förderband Zuführung Vereinzler   AST*)
ST03_425_B67_1(ValveObject:= ADR(ST03_426_Y68_5));(*Förderband Zuführung Vereinzler   GST*)

(* Call ST03_426_Y68_6 Förderband  Zuführung Stopper AST/GST  (Valve) *)
Analyze(InputExp:=  TRUE, DoAnalyze:= TRUE );
ST03_426_Y68_6.strAnlayse:=Analyze.OutString;
ST03_426_Y68_6(Enable  :=  Analyze.ExpResult,
                                sVisu:=Visu.ST03_426_Y68_6,
                                Reset:=gResetAll,
);
ST03_425_B67_2(ValveObject:= ADR(ST03_426_Y68_6));(*Förderband Zuführung Stopper   AST*)
ST03_425_B67_3(ValveObject:= ADR(ST03_426_Y68_6));(*Förderband Zuführung Stopper   GST*)

(* Call ST03_425_B67_4 Zuführung  frei zum Ablegen ISK SP Maschine Pos.1  (DigIn) *)
ST03_425_B67_4(sVisu:=Visu.ST03_425_B67_4,
                                Reset:=gResetAll,
);
(* Call ST03_425_B67_5 Zuführung  frei zum Ablegen ISK SP Maschine Pos.2  (DigIn) *)
ST03_425_B67_5(sVisu:=Visu.ST03_425_B67_5,
                                Reset:=gResetAll,
);
(* Call ST03_425_B67_6 Zuführung  frei zum Ablegen ISK SP Maschine Pos.3  (DigIn) *)
ST03_425_B67_6(sVisu:=Visu.ST03_425_B67_6,
                                Reset:=gResetAll,
);
(* Call ST03_425_B67_7 Zuführung  frei zum Ablegen ISK SP Maschine Pos.3  (DigIn) *)
ST03_425_B67_7(sVisu:=Visu.ST03_425_B67_7,
                                Reset:=gResetAll,
);
(* Call ST03_426_B68_4  ISK anwesend am Vereinzler  (DigIn) *)
ST03_426_B68_4(sVisu:=Visu.ST03_426_B68_4,
                                Reset:=gResetAll,
);
END_ACTION
ACTION call_154polRP:
(* Call ST03_418_B60_6 Zuführung links frei zum Ablegen ISK SP Maschine (DigIn) *)
ST03_418_B60_6(sVisu:=Visu.ST03_418_B60_6,
                                Reset:=gResetAll,
);
(* Call ST03_418_B60_7 Zuführung rechts frei zum Ablegen ISK SP Maschine (DigIn) *)
ST03_418_B60_7(sVisu:=Visu.ST03_418_B60_7,
                                Reset:=gResetAll,
);
(* Call ST03_419_B61_0 Förderband Zuführung links ISK anwesend zum Vereinzeln (DigIn) *)
ST03_419_B61_0(sVisu:=Visu.ST03_419_B61_0,
                                Reset:=gResetAll,
);
(* Call ST03_419_B61_1 Förderband Zuführung rechts ISK anwesend zum Vereinzeln (DigIn) *)
ST03_419_B61_1(sVisu:=Visu.ST03_419_B61_1,
                                Reset:=gResetAll,
);
(* Call ST03_419_B61_2 Züführung links ISK auf Übergabeposition Roboter Palettierer (DigIn) *)
ST03_419_B61_2(sVisu:=Visu.ST03_419_B61_2,
                                Reset:=gResetAll,
);
(* Call ST03_419_B61_3 Züführung rechts ISK auf Übergabeposition Roboter Palettierer (DigIn) *)
ST03_419_B61_3(sVisu:=Visu.ST03_419_B61_3,
                                Reset:=gResetAll,
);
(* Call ST03_419_Y61_5 Förderband linke Zuführung Vereinzler AST/GST  (Valve) *)
Analyze(InputExp:=  TRUE, DoAnalyze:= TRUE );
ST03_419_Y61_5.strAnlayse:=Analyze.OutString;
ST03_419_Y61_5(Enable  :=  Analyze.ExpResult,
                                sVisu:=Visu.ST03_419_Y61_5,
                                Reset:=gResetAll,
);
ST03_418_B60_0(ValveObject:= ADR(ST03_419_Y61_5));(*  Förderband linke Zuführung Vereinzler AST*)
ST03_418_B60_1(ValveObject:= ADR(ST03_419_Y61_5));(*  Förderband linke Zuführung Vereinzler GST*)

(* Call ST03_419_Y61_6 Förderband rechte Zuführung Vereinzler AST/GST  (Valve) *)
Analyze(InputExp:=  TRUE, DoAnalyze:= TRUE );
ST03_419_Y61_6.strAnlayse:=Analyze.OutString;
ST03_419_Y61_6(Enable  :=  Analyze.ExpResult,
                                sVisu:=Visu.ST03_419_Y61_6,
                                Reset:=gResetAll,
);
ST03_418_B60_2(ValveObject:= ADR(ST03_419_Y61_6));(*Förderband rechte Zuführung Vereinzler   AST*)
ST03_418_B60_3(ValveObject:= ADR(ST03_419_Y61_6));(*Förderband rechte Zuführung Vereinzler   GST*)

(* Call ST03_419_Y61_7 Förderband links/rechts Züführung Stopper AST/GST  (Valve) *)
Analyze(InputExp:=  TRUE, DoAnalyze:= TRUE );
ST03_419_Y61_7.strAnlayse:=Analyze.OutString;
ST03_419_Y61_7(Enable  :=  Analyze.ExpResult,
                                sVisu:=Visu.ST03_419_Y61_7,
                                Reset:=gResetAll,
);
ST03_418_B60_4(ValveObject:= ADR(ST03_419_Y61_7));(*Förderband links/rechts Zuführung Stopper   AST*)
ST03_418_B60_5(ValveObject:= ADR(ST03_419_Y61_7));(*Förderband links/rechts Zuführung Stopper   GST*)
END_ACTION
ACTION call_191pol:
(* Call ST03_541_B69_0 IZuführung  frei zum Ablegen ISK SP Maschine (DigIn) *)
ST03_541_B69_0(sVisu:=Visu.ST03_541_B69_0,
                                Reset:=gResetAll,
);
(* Call ST03_542_Y70_1  Zuführung Vereinzler AST/GST  (Valve) *)
Analyze(InputExp:=  TRUE, DoAnalyze:= TRUE );
ST03_542_Y70_1.strAnlayse:=Analyze.OutString;
ST03_542_Y70_1(Enable  :=  Analyze.ExpResult,
                                sVisu:=Visu.ST03_542_Y70_1,
                                Reset:=gResetAll,
);
ST03_541_B69_1(ValveObject:= ADR(ST03_542_Y70_1));(*  Zuführung Vereinzler eingefahren GST*)
ST03_541_B69_2(ValveObject:= ADR(ST03_542_Y70_1));(*  Zuführung Vereinzler ausgefahren AST*)

(* Call ST03_542_Y70_2  Züführung Stopper AST/GST  (Valve) *)
Analyze(InputExp:=  TRUE, DoAnalyze:= TRUE );
ST03_542_Y70_2.strAnlayse:=Analyze.OutString;
ST03_542_Y70_2(Enable  :=  Analyze.ExpResult,
                                sVisu:=Visu.ST03_542_Y70_2,
                                Reset:=gResetAll,
);
ST03_541_B69_3(ValveObject:= ADR(ST03_542_Y70_2));(* Zuführung Stopper  eingefahren  AST*)
ST03_541_B69_4(ValveObject:= ADR(ST03_542_Y70_2));(* Zuführung Stopper  ausgefahren GST*)


(* Call ST03_541_B69_6 SK anwesend am Stoper (DigIn) *)
ST03_541_B69_6(sVisu:=Visu.ST03_541_B69_6,
                                Reset:=gResetAll,
);
(* Call ST03_541_B69_7  ISK Lageerkennung links (DigIn) *)
ST03_541_B69_7(sVisu:=Visu.ST03_541_B69_7,
                                Reset:=gResetAll,
);
(* Call ST03_542_B70_0  ISK Lageerkennung rechts (DigIn) *)
ST03_542_B70_0(sVisu:=Visu.ST03_542_B70_0,
                                Reset:=gResetAll,
);
END_ACTION
ACTION call_206pol:
(* Call ST03_437_Y68_5 Förderband  Zuführung Vereinzler AST/GST  (Valve) *)
Analyze(InputExp:=  TRUE, DoAnalyze:= TRUE );
ST03_437_Y68_5.strAnlayse:=Analyze.OutString;
ST03_437_Y68_5(Enable  :=  Analyze.ExpResult,
                                sVisu:=Visu.ST03_437_Y68_5,
                                Reset:=gResetAll,
);
ST03_435_B67_0(ValveObject:= ADR(ST03_437_Y68_5));(*Förderband Zuführung Vereinzler   AST*)
ST03_435_B67_1(ValveObject:= ADR(ST03_437_Y68_5));(*Förderband Zuführung Vereinzler   GST*)

(* Call ST03_426_Y68_6 Förderband  Zuführung Stopper AST/GST  (Valve) *)
Analyze(InputExp:=  TRUE, DoAnalyze:= TRUE );
ST03_437_Y68_6.strAnlayse:=Analyze.OutString;
ST03_437_Y68_6(Enable  :=  Analyze.ExpResult,
                                sVisu:=Visu.ST03_437_Y68_6,
                                Reset:=gResetAll,
);
ST03_435_B67_2(ValveObject:= ADR(ST03_437_Y68_6));(*Förderband Zuführung Stopper   AST*)
ST03_435_B67_3(ValveObject:= ADR(ST03_437_Y68_6));(*Förderband Zuführung Stopper   GST*)

(* Call ST03_435_B67_4 Zuführung  frei zum Ablegen ISK SP Maschine Pos.1  (DigIn) *)
ST03_435_B67_4(sVisu:=Visu.ST03_435_B67_4,
                                Reset:=gResetAll,
);
(* Call ST03_435_B67_7 Zuführung  ISK anwesend am Stopper (DigIn) *)
ST03_435_B67_7(sVisu:=Visu.ST03_435_B67_7,
                                Reset:=gResetAll,
);
(* Call ST03_437_B68_4  ISK auf Übergabeposition zu Roboterr  (DigIn) *)
ST03_437_B68_4(sVisu:=Visu.ST03_437_B68_4,
                                Reset:=gResetAll,
);
(* Call ST03_436_B68_1 Zuführung  ISK Lageerkennung links (DigIn) *)
ST03_436_B68_1(sVisu:=Visu.ST03_436_B68_1,
                                Reset:=gResetAll,
);
(* Call ST03_436_B68_2 Zuführung  ISK Lageerkennung links (DigIn) *)
ST03_436_B68_2(sVisu:=Visu.ST03_436_B68_2,
                                Reset:=gResetAll,
);
END_ACTION
ACTION call_21pol:
(* Call ST03_536_B69_0 IZuführung  frei zum Ablegen ISK SP Maschine (DigIn) *)
ST03_536_B69_0(sVisu:=Visu.ST03_536_B69_0,
                                Reset:=gResetAll,
);
(* Call ST03_537_Y70_1  Zuführung Vereinzler AST/GST  (Valve) *)
Analyze(InputExp:=  TRUE, DoAnalyze:= TRUE );
ST03_537_Y70_1.strAnlayse:=Analyze.OutString;
ST03_537_Y70_1(Enable  :=  Analyze.ExpResult,
                                sVisu:=Visu.ST03_537_Y70_1,
                                Reset:=gResetAll,
);
ST03_536_B69_1(ValveObject:= ADR(ST03_537_Y70_1));(*  Zuführung Vereinzler eingefahren GST*)
ST03_536_B69_2(ValveObject:= ADR(ST03_537_Y70_1));(*  Zuführung Vereinzler ausgefahren AST*)

(* Call ST03_537_Y70_2  Züführung Stopper AST/GST  (Valve) *)
Analyze(InputExp:=  TRUE, DoAnalyze:= TRUE );
ST03_537_Y70_2.strAnlayse:=Analyze.OutString;
ST03_537_Y70_2(Enable  :=  Analyze.ExpResult,
                                sVisu:=Visu.ST03_537_Y70_2,
                                Reset:=gResetAll,
);
ST03_536_B69_3(ValveObject:= ADR(ST03_537_Y70_2));(* Zuführung Stopper  eingefahren  AST*)
ST03_536_B69_4(ValveObject:= ADR(ST03_537_Y70_2));(* Zuführung Stopper  ausgefahren GST*)


(* Call ST03_536_B69_6 SK anwesend am Stoper (DigIn) *)
ST03_536_B69_6(sVisu:=Visu.ST03_536_B69_6,
                                Reset:=gResetAll,
);
(* Call ST03_536_B69_7 ISK anwesend an Abholposition (DigIn) *)
ST03_536_B69_7(sVisu:=Visu.ST03_536_B69_7,
                                Reset:=gResetAll,
);
(* Call ST03_537_B70_0  ISK Lageerkennung (DigIn) *)
ST03_537_B70_0(sVisu:=Visu.ST03_537_B70_0,
                                Reset:=gResetAll,
);
END_ACTION
ACTION call_268pol_102pol_neu:
ST03_8_100_A1(
		Activated := MP.ST03.CamOn[1],
		st_InstName:='ST03_8_100_A1',
		st_Description:= 'Kamera 1 Farberkennung',
		SensopartErgebnis:=TD.SensopartErgebnis,
		);
ST03_8_100_A1.s_IpAdress := MP.ST03.SensopartIPAdress[1];  		(* 'MP.SensopartIPAdress';*)
ST03_8_100_A1.i_CmdPort := 2006;
ST03_8_100_A1.i_DataPort :=2005;

IF	gTypeCode = 4993 THEN
	ST03_8_103_A1(
			Activated := MP.ST03.CamOn[2],
			st_InstName:='ST03_8_103_A1',
			st_Description:= 'Kamera 2 Flügelerkennung',
			SensopartErgebnis:=TD.Sensopart2Ergebnis,
			);
	ST03_8_103_A1.s_IpAdress := MP.ST03.SensopartIPAdress[2];  		(* 'MP.SensopartIPAdress';*)
	ST03_8_103_A1.i_CmdPort := 2006;
	ST03_8_103_A1.i_DataPort :=2005;
END_IF


(* Call ST03_556_B69_0 IZuführung  frei zum Ablegen ISK SP Maschine (DigIn) *)
ST03_556_B69_0(sVisu:=Visu.ST03_556_B69_0,
                                Reset:=gResetAll,
);
(* Call ST03_556_Y70_1  Zuführung Vereinzler AST/GST  (Valve) *)
Analyze(InputExp:=  TRUE, DoAnalyze:= TRUE );
ST03_557_Y70_1.strAnlayse:=Analyze.OutString;
ST03_557_Y70_1(Enable  :=  Analyze.ExpResult,
                                sVisu:=Visu.ST03_557_Y70_1,
                                Reset:=gResetAll,
);
ST03_556_B69_1(ValveObject:= ADR(ST03_557_Y70_1));(*  Zuführung Vereinzler eingefahren GST*)
ST03_556_B69_2(ValveObject:= ADR(ST03_557_Y70_1));(*  Zuführung Vereinzler ausgefahren AST*)

(* Call ST03_556_Y70_2  Züführung Stopper AST/GST  (Valve) *)
Analyze(InputExp:=  TRUE, DoAnalyze:= TRUE );
ST03_557_Y70_2.strAnlayse:=Analyze.OutString;
ST03_557_Y70_2(Enable  :=  Analyze.ExpResult,
                                sVisu:=Visu.ST03_557_Y70_2,
                                Reset:=gResetAll,
);
ST03_556_B69_3(ValveObject:= ADR(ST03_557_Y70_2));(* Zuführung Stopper  eingefahren  AST*)
ST03_556_B69_4(ValveObject:= ADR(ST03_557_Y70_2));(* Zuführung Stopper  ausgefahren GST*)

(* Call ST03_556_B69_5 Führungsschiene Überwachung Staustrecke (DigIn) *)
ST03_556_B69_5(sVisu:=Visu.ST03_556_B69_5,
                                Reset:=gResetAll,
);

(* Call ST03_556_B69_6 SK anwesend am Stoper (DigIn) *)
ST03_556_B69_6(sVisu:=Visu.ST03_556_B69_6,
                                Reset:=gResetAll,
);
(* Call ST03_546_B69_7 ISK  auf Übergabeposition  (DigIn) *)
ST03_556_B69_7(sVisu:=Visu.ST03_556_B69_7,
                                Reset:=gResetAll,
);
END_ACTION
ACTION call_268polRP:
(*Rüstsatz 268 pol Rasterplatte======================================================================================*)

(* Call ST03_562_B69_0 Zuführung 1 frei zum schwenken (DigIn) *)
ST03_562_B69_0(sVisu:=Visu.ST03_562_B69_0,
                                Reset:=gResetAll,
);
(* Call ST03_562_B69_6 Zuführung 1 ISK anwesend am Stopper (DigIn) *)
ST03_562_B69_6(sVisu:=Visu.ST03_562_B69_6,
                                Reset:=gResetAll,
);
(* Call ST03_562_B67_7 Zuführung 1 ISK auf Übergabepos. Robi (DigIn) *)
ST03_562_B67_7(sVisu:=Visu.ST03_562_B67_7,
                                Reset:=gResetAll,
);
(* Call ST03_563_B70_0 Zuführung 2 frei zum schwenken (DigIn) *)
ST03_563_B70_0(sVisu:=Visu.ST03_563_B70_0,
                                Reset:=gResetAll,
);
(* Call ST03_563_B70_6 Zuführung 2 ISK anwesend am Stopper (DigIn) *)
ST03_563_B70_6(sVisu:=Visu.ST03_563_B70_6,
                                Reset:=gResetAll,
);
(* Call ST03_563_B70_7 Zuführung 2 ISK auf Übergabepos. Robi (DigIn) *)
ST03_563_B70_7(sVisu:=Visu.ST03_563_B70_7,
                                Reset:=gResetAll,
);
(* Call ST03_565_B72_0 ISK 1 in Klemmer (DigIn) *)
ST03_565_B72_0(sVisu:=Visu.ST03_565_B72_0,
                                Reset:=gResetAll,
);
(* Call ST03_565_B72_1 ISK 2 in Klemmer (DigIn) *)
ST03_565_B72_1(sVisu:=Visu.ST03_565_B72_1,
                                Reset:=gResetAll,
);
(* Call ST03_564_Y71_0 Zuführung 1 Vereinzler AST/GST  (Valve) *)
Analyze(InputExp:=  TRUE, DoAnalyze:= TRUE );
ST03_564_Y71_0.strAnlayse:=Analyze.OutString;
ST03_564_Y71_0(Enable  :=  Analyze.ExpResult,
                                sVisu:=Visu.ST03_564_Y71_0,
                                Reset:=gResetAll,
);
ST03_562_B69_1(ValveObject:= ADR(ST03_564_Y71_0));(*Zuführung 1 Zuführung Vereinzler AST*)
ST03_562_B69_2(ValveObject:= ADR(ST03_564_Y71_0));(*Zuführung 1 Zuführung Vereinzler GST*)

(* Call ST03_564_Y71_1 Zuführung 1 Stopper AST/GST  (Valve) *)
Analyze(InputExp:=  TRUE, DoAnalyze:= TRUE );
ST03_564_Y71_1.strAnlayse:=Analyze.OutString;
ST03_564_Y71_1(Enable  :=  Analyze.ExpResult,
                                sVisu:=Visu.ST03_564_Y71_1,
                                Reset:=gResetAll,
);
ST03_562_B69_3(ValveObject:= ADR(ST03_564_Y71_1));(*Zuführung 1 Zuführung Stopper AST*)
ST03_562_B69_4(ValveObject:= ADR(ST03_564_Y71_1));(*Zuführung 1 Zuführung Stopper GST*)

(* Call ST03_564_Y71_2 Zuführung 2 Vereinzler AST/GST  (Valve) *)
Analyze(InputExp:=  TRUE, DoAnalyze:= TRUE );
ST03_564_Y71_2.strAnlayse:=Analyze.OutString;
ST03_564_Y71_2(Enable  :=  Analyze.ExpResult,
                                sVisu:=Visu.ST03_564_Y71_2,
                                Reset:=gResetAll,
);
ST03_563_B70_1(ValveObject:= ADR(ST03_564_Y71_2));(*Zuführung 2 Zuführung Vereinzler AST*)
ST03_563_B70_2(ValveObject:= ADR(ST03_564_Y71_2));(*Zuführung 2 Zuführung Vereinzler GST*)

(* Call ST03_564_Y71_3 Zuführung 2 Stopper AST/GST  (Valve) *)
Analyze(InputExp:=  TRUE, DoAnalyze:= TRUE );
ST03_564_Y71_3.strAnlayse:=Analyze.OutString;
ST03_564_Y71_3(Enable  :=  Analyze.ExpResult,
                                sVisu:=Visu.ST03_564_Y71_3,
                                Reset:=gResetAll,
);
ST03_563_B70_3(ValveObject:= ADR(ST03_564_Y71_3));(*Zuführung 2 Zuführung Stopper AST*)
ST03_563_B70_4(ValveObject:= ADR(ST03_564_Y71_3));(*Zuführung 2 Zuführung Stopper GST*)


(* Call ST03_564_Y71_4 ISK Klemmer  AST/GST  (Valve) *)
Analyze(InputExp:=  TRUE, DoAnalyze:= TRUE );
ST03_564_Y71_4.strAnlayse:=Analyze.OutString;
ST03_564_Y71_4(Enable  :=  Analyze.ExpResult,
                                sVisu:=Visu.ST03_564_Y71_4,
                                Reset:=gResetAll,
);
ST03_565_B72_4(ValveObject:= ADR(ST03_564_Y71_4));(*ISK Klemmer 2 offen GST*)
ST03_565_B72_5(ValveObject:= ADR(ST03_564_Y71_4));(*ISK Klemmer 2 zu AST*)
ST03_565_B72_2(ValveObject:= ADR(ST03_564_Y71_4));(*ISK Klemmer 1 offen GST*)
ST03_565_B72_3(ValveObject:= ADR(ST03_564_Y71_4));(*ISK Klemmer 1 zu AST*)

(* Call ST03_564_Y71_5 Rinne schwenkern AST/GST  (Valve) *)
Analyze(InputExp:=  TRUE, DoAnalyze:= TRUE );
ST03_564_Y71_5.strAnlayse:=Analyze.OutString;
ST03_564_Y71_5(Enable  :=  Analyze.ExpResult,
                                sVisu:=Visu.ST03_564_Y71_5,
                                Reset:=gResetAll,
);
ST03_565_B72_6(ValveObject:= ADR(ST03_564_Y71_5));(*ISK Klemmer schwenkern 0° AST*)
ST03_565_B72_7(ValveObject:= ADR(ST03_564_Y71_5));(*ISK Klemmer schwenkern 180° GST*)
END_ACTION
ACTION call_33pol:
(* Call ST03_571_B69_0 Zuführung Pos 1  frei zum Ablegen ISK SP Maschine (DigIn) *)
ST03_571_B69_0(sVisu:=Visu.ST03_571_B69_0,
                                Reset:=gResetAll,
);
(* Call ST03_571_B69_1 Zuführung Pos 2  frei zum Ablegen ISK SP Maschine (DigIn) *)
ST03_571_B69_1(sVisu:=Visu.ST03_571_B69_1,
                                Reset:=gResetAll,
);

(* Call ST03_572_Y70_0  Zuführung Vereinzler AST/GST  (Valve) *)
Analyze(InputExp:=  TRUE, DoAnalyze:= TRUE );
ST03_572_Y70_0.strAnlayse:=Analyze.OutString;
ST03_572_Y70_0(Enable  :=  Analyze.ExpResult,
                                sVisu:=Visu.ST03_572_Y70_0,
                                Reset:=gResetAll,
);
ST03_571_B69_2(ValveObject:= ADR(ST03_572_Y70_0));(*  Zuführung Vereinzler eingefahren GST*)
ST03_571_B69_3(ValveObject:= ADR(ST03_572_Y70_0));(*  Zuführung Vereinzler ausgefahren AST*)

(* Call ST03_572_Y70_1  Züführung Stopper AST/GST  (Valve) *)
Analyze(InputExp:=  TRUE, DoAnalyze:= TRUE );
ST03_572_Y70_1.strAnlayse:=Analyze.OutString;
ST03_572_Y70_1(Enable  :=  Analyze.ExpResult,
                                sVisu:=Visu.ST03_572_Y70_1,
                                Reset:=gResetAll,
);
ST03_571_B69_4(ValveObject:= ADR(ST03_572_Y70_1));(* Zuführung Stopper  eingefahren  AST*)
ST03_571_B69_5(ValveObject:= ADR(ST03_572_Y70_1));(* Zuführung Stopper  ausgefahren GST*)


(* Call ST03_571_B69_6 SK anwesend am Stoper (DigIn) *)
ST03_571_B69_6(sVisu:=Visu.ST03_571_B69_6,
                                Reset:=gResetAll,
);
(* Call ST03_571_B69_7 ISK anwesend an Abholposition (DigIn) *)
ST03_571_B69_7(sVisu:=Visu.ST03_571_B69_7,
                                Reset:=gResetAll,
);
END_ACTION
ACTION call_46pol:
(* Call ST03_463_Y71_3 Förderband  Zuführung Vereinzler AST/GST  (Valve) *)
Analyze(InputExp:=  TRUE, DoAnalyze:= TRUE );
ST03_464_Y71_3.strAnlayse:=Analyze.OutString;
ST03_464_Y71_3(Enable  :=  Analyze.ExpResult,
                                sVisu:=Visu.ST03_464_Y71_3,
                                Reset:=gResetAll,
);
ST03_461_B69_0(ValveObject:= ADR(ST03_464_Y71_3));(*Förderband Zuführung Vereinzler   AST*)
ST03_461_B69_1(ValveObject:= ADR(ST03_464_Y71_3));(*Förderband Zuführung Vereinzler   GST*)

(* Call ST03_463_Y71_4 Förderband  Zuführung Stopper AST/GST  (Valve) *)
Analyze(InputExp:=  TRUE, DoAnalyze:= TRUE );
ST03_464_Y71_4.strAnlayse:=Analyze.OutString;
ST03_464_Y71_4(Enable  :=  Analyze.ExpResult,
                                sVisu:=Visu.ST03_464_Y71_4,
                                Reset:=gResetAll,
);
ST03_461_B69_2(ValveObject:= ADR(ST03_464_Y71_4));(*Förderband Zuführung Stopper   AST*)
ST03_461_B69_3(ValveObject:= ADR(ST03_464_Y71_4));(*Förderband Zuführung Stopper   GST*)

(* Call ST03_461_B69_4 Zuführung  frei zum Ablegen ISK SP Maschine Pos.1  (DigIn) *)
ST03_461_B69_4(sVisu:=Visu.ST03_461_B69_4,
                                Reset:=gResetAll,
);
(* Call ST03_461_B69_7 Zuführung  ISK anwesend am Stopper (DigIn) *)
ST03_461_B69_7(sVisu:=Visu.ST03_461_B69_7,
                                Reset:=gResetAll,
);
(* Call ST03_463_B70_7  ISK auf Übergabeposition zu Roboter  (DigIn) *)
ST03_463_B70_7(sVisu:=Visu.ST03_463_B70_7,
                                Reset:=gResetAll,
);
(* Call ST03_462_B70_0 Förderband  ISK anwesend Wender (DigIn) *)
ST03_462_B70_0(sVisu:=Visu.ST03_462_B70_0,
                                Reset:=gResetAll,
);
(* Call ST03_462_B70_1 Zuführung  ISK Lageerkennung rechts (DigIn) *)
ST03_462_B70_1(sVisu:=Visu.ST03_462_B70_1,
                                Reset:=gResetAll,
);
(* Call ST03_462_B70_2 Zuführung  ISK Lageerkennung links (DigIn) *)
ST03_462_B70_2(sVisu:=Visu.ST03_462_B70_2,
                                Reset:=gResetAll,
);
(* Call ST03_464_Y71_0 Förderband  Zuführung Vereinzelner Wender AST/GST  (Valve) *)
Analyze(InputExp:=  TRUE, DoAnalyze:= TRUE );
ST03_464_Y71_0.strAnlayse:=Analyze.OutString;
ST03_464_Y71_0(Enable  :=  Analyze.ExpResult,
                                sVisu:=Visu.ST03_464_Y71_0,
                                Reset:=gResetAll,
);
ST03_461_B69_5(ValveObject:= ADR(ST03_464_Y71_0));(*Förderbandeinheit  Zuführung  Vereinzelner Wender AST*)
ST03_461_B69_6(ValveObject:= ADR(ST03_464_Y71_0));(*Förderbandeinheit  Zuführung  Vereinzelner Wender GST*)

(* Call ST03_464_Y71_1 Förderband  Zuführung Zylinder Vakuumdüsen AST/GST  (Valve) *)
Analyze(InputExp:=  TRUE, DoAnalyze:= TRUE );
ST03_464_Y71_1.strAnlayse:=Analyze.OutString;
ST03_464_Y71_1(Enable  :=  Analyze.ExpResult,
                                sVisu:=Visu.ST03_464_Y71_1,
                                Reset:=gResetAll,
);
ST03_463_B70_3(ValveObject:= ADR(ST03_464_Y71_1));(*Förderband Zuführung Zylinder Vakuumdüsen   AST*)
ST03_463_B70_4(ValveObject:= ADR(ST03_464_Y71_1));(*Förderband Zuführung Zylinder Vakuumdüsen   GST*)

IF	ST03_463_B70_3.ValveSensor THEN
	ST03_463_B70_3_4_pos:= -14;
ELSIF
	ST03_463_B70_4.ValveSensor THEN
	ST03_463_B70_3_4_pos:= 0;
ELSE
	ST03_463_B70_3_4_pos:= -7;
END_IF

(* Call ST03_464_Y71_2  Förderband  Zuführung Wendestation Einlauf / Auslauf   (Valve) *)
Analyze(InputExp:=  TRUE, DoAnalyze:= TRUE );
ST03_464_Y71_2.strAnlayse:=Analyze.OutString;
ST03_464_Y71_2(Enable  :=  Analyze.ExpResult,
                                sVisu:=Visu.ST03_464_Y71_2,
                                Reset:=gResetAll,
);
ST03_463_B70_5(ValveObject:= ADR(ST03_464_Y71_2));(*Förderband Zuführung Wendestation   AST*)
ST03_463_B70_6(ValveObject:= ADR(ST03_464_Y71_2));(*Förderband Zuführung Wendestation   GST*)

(* Call ST03_464_Y71_5  Förderband  Zuführung Vakuumdüsen EIN/AUS  (Valve) *)
Analyze(InputExp:=  TRUE, DoAnalyze:= TRUE );
ST03_464_Y71_5.strAnlayse:=Analyze.OutString;
ST03_464_Y71_5(Enable  :=  Analyze.ExpResult,
                                sVisu:=Visu.ST03_464_Y71_5,
                                Reset:=gResetAll,
);
(* Call ST03_464_B71_6  Vakuum vorhanden (DigIn) *)
ST03_464_B71_6(sVisu:=Visu.ST03_464_B71_6,
                                Reset:=gResetAll,
);
(* Call ST03_464_B71_7 Förderband  Staustrecke mitte voll (DigIn) *)
ST03_464_B71_7(sVisu:=Visu.ST03_464_B71_7,
                                Reset:=gResetAll,
);
END_ACTION
ACTION call_48pol:
(* Call ST03_551_B69_0 IZuführung  frei zum Ablegen ISK SP Maschine (DigIn) *)
ST03_551_B69_0(sVisu:=Visu.ST03_551_B69_0,
                                Reset:=gResetAll,
);
(* Call ST03_552_Y70_1  Zuführung Vereinzler AST/GST  (Valve) *)
Analyze(InputExp:=  TRUE, DoAnalyze:= TRUE );
ST03_552_Y70_1.strAnlayse:=Analyze.OutString;
ST03_552_Y70_1(Enable  :=  Analyze.ExpResult,
                                sVisu:=Visu.ST03_552_Y70_1,
                                Reset:=gResetAll,
);
ST03_551_B69_1(ValveObject:= ADR(ST03_552_Y70_1));(*  Zuführung Vereinzler eingefahren GST*)
ST03_551_B69_2(ValveObject:= ADR(ST03_552_Y70_1));(*  Zuführung Vereinzler ausgefahren AST*)

(* Call ST03_552_Y70_2  Züführung Stopper AST/GST  (Valve) *)
Analyze(InputExp:=  TRUE, DoAnalyze:= TRUE );
ST03_552_Y70_2.strAnlayse:=Analyze.OutString;
ST03_552_Y70_2(Enable  :=  Analyze.ExpResult,
                                sVisu:=Visu.ST03_552_Y70_2,
                                Reset:=gResetAll,
);
ST03_551_B69_3(ValveObject:= ADR(ST03_552_Y70_2));(* Zuführung Stopper  eingefahren  AST*)
ST03_551_B69_4(ValveObject:= ADR(ST03_552_Y70_2));(* Zuführung Stopper  ausgefahren GST*)


(* Call ST03_551_B69_6 SK anwesend am Stoper (DigIn) *)
ST03_551_B69_6(sVisu:=Visu.ST03_551_B69_6,
                                Reset:=gResetAll,
);
(* Call ST03_541_B69_7 ISK Lageerkennung links (DigIn) *)
ST03_551_B69_7(sVisu:=Visu.ST03_551_B69_7,
                                Reset:=gResetAll,
);
(* Call ST03_542_B70_0  ISK Lageerkennung rechts (DigIn) *)
ST03_552_B70_0(sVisu:=Visu.ST03_552_B70_0,
                                Reset:=gResetAll,
);
END_ACTION
ACTION call_72pol:
(* Call ST03_546_B69_0 IZuführung  frei zum Ablegen ISK SP Maschine (DigIn) *)
ST03_546_B69_0(sVisu:=Visu.ST03_546_B69_0,
                                Reset:=gResetAll,
);
(* Call ST03_547_Y70_1  Zuführung Vereinzler AST/GST  (Valve) *)
Analyze(InputExp:=  TRUE, DoAnalyze:= TRUE );
ST03_547_Y70_1.strAnlayse:=Analyze.OutString;
ST03_547_Y70_1(Enable  :=  Analyze.ExpResult,
                                sVisu:=Visu.ST03_547_Y70_1,
                                Reset:=gResetAll,
);
ST03_546_B69_1(ValveObject:= ADR(ST03_547_Y70_1));(*  Zuführung Vereinzler eingefahren GST*)
ST03_546_B69_2(ValveObject:= ADR(ST03_547_Y70_1));(*  Zuführung Vereinzler ausgefahren AST*)

(* Call ST03_547_Y70_2  Züführung Stopper AST/GST  (Valve) *)
Analyze(InputExp:=  TRUE, DoAnalyze:= TRUE );
ST03_547_Y70_2.strAnlayse:=Analyze.OutString;
ST03_547_Y70_2(Enable  :=  Analyze.ExpResult,
                                sVisu:=Visu.ST03_547_Y70_2,
                                Reset:=gResetAll,
);
ST03_546_B69_3(ValveObject:= ADR(ST03_547_Y70_2));(* Zuführung Stopper  eingefahren  AST*)
ST03_546_B69_4(ValveObject:= ADR(ST03_547_Y70_2));(* Zuführung Stopper  ausgefahren GST*)


(* Call ST03_546_B69_6 SK anwesend am Stoper (DigIn) *)
ST03_546_B69_6(sVisu:=Visu.ST03_546_B69_6,
                                Reset:=gResetAll,
);
(* Call ST03_546_B69_7 ISK anwesend an Abholposition (DigIn) *)
ST03_546_B69_7(sVisu:=Visu.ST03_546_B69_7,
                                Reset:=gResetAll,
);
(* Call ST03_547_B70_0  ISK Lageerkennung (DigIn) *)
ST03_547_B70_0(sVisu:=Visu.ST03_547_B70_0,
                                Reset:=gResetAll,
);
END_ACTION
ACTION call_74_91_35_168_160pol:
(* Call ST03_421_B63_4 Förderband frei zum Ablegen ISK SP Maschine Pos1  (DigIn) *)
ST03_421_B63_4(sVisu:=Visu.ST03_421_B63_4,
                                Reset:=gResetAll,
);
(* Call ST03_421_B63_5 Förderband frei zum Ablegen ISK SP Maschine Pos2  (DigIn) *)
ST03_421_B63_5(sVisu:=Visu.ST03_421_B63_5,
                                Reset:=gResetAll,
);
(* Call ST03_421_B63_6 Förderband frei zum Ablegen ISK SP Maschine Pos3  (DigIn) *)
ST03_421_B63_6(sVisu:=Visu.ST03_421_B63_6,
                                Reset:=gResetAll,
);
(* Call ST03_421_B63_7 ISK anwesend am Vereinzler  (DigIn) *)
ST03_421_B63_7(sVisu:=Visu.ST03_421_B63_7,
                                Reset:=gResetAll,
);
(* Call ST03_422_B64_0 Förderband Trigger Tintenstrahldrucker (Lichtschranke)  (DigIn) *)
ST03_422_B64_0(sVisu:=Visu.ST03_422_B64_0,
                                Reset:=gResetAll,
);
(* Call ST03_423_B66_0 Förderband Trigger Tintenstrahldrucker (Lichtschranke)  (DigIn) *)
ST03_423_B66_0(sVisu:=Visu.ST03_423_B66_0,
                                Reset:=gResetAll,
);
(* Call ST03_8_B76_1 Förderband Trigger Tintenstrahldrucker (Lichtschranke)  (DigIn) 3621 *)
ST03_8_B76_1(sVisu:=Visu.ST03_8_B76_1,
                                Reset:=gResetAll,
);
(* Call ST03_8_B76_2 Förderband Trigger Tintenstrahldrucker (Lichtschranke)  (DigIn) 3621 *)
ST03_8_B76_2(sVisu:=Visu.ST03_8_B76_2,
                                Reset:=gResetAll,
);
(* Call ST03_422_B64_3  Förderband ISK anwesend Stopper Kamera  (DigIn) *)
ST03_422_B64_3(sVisu:=Visu.ST03_422_B64_3,
                                Reset:=gResetAll,
);
(* Call ST03_422_B64_4 Zuführung ISK auf Übergabeposition Robo Palettierer  (DigIn) *)
ST03_422_B64_4(sVisu:=Visu.ST03_422_B64_4,
                                Reset:=gResetAll,
);
(* Call ST03_422_Y64_5  Förderband  Zuführung Vereinzler AST/GST (Valve) *)
Analyze(InputExp:=  TRUE, DoAnalyze:= TRUE );
ST03_422_Y64_5.strAnlayse:=Analyze.OutString;
ST03_422_Y64_5(Enable  :=  Analyze.ExpResult,
                                sVisu:=Visu.ST03_422_Y64_5,
                                Reset:=gResetAll,
);
ST03_421_B63_0(ValveObject:= ADR(ST03_422_Y64_5));(*Förderband Zuführung Vereinzler AST*)
ST03_421_B63_1(ValveObject:= ADR(ST03_422_Y64_5));(*Förderband Zuführung Vereinzler GST*)

(* Call ST03_422_Y64_6 Förderband rechte Zuführung Vereinzler AST/GST (Valve) *)
Analyze(InputExp:=  TRUE, DoAnalyze:= TRUE );
ST03_422_Y64_6.strAnlayse:=Analyze.OutString;
ST03_422_Y64_6(Enable  :=  Analyze.ExpResult,
                                sVisu:=Visu.ST03_422_Y64_6,
                                Reset:=gResetAll,
);
ST03_421_B63_2(ValveObject:= ADR(ST03_422_Y64_6));(*Förderband Zuführung Stopper AST*)
ST03_421_B63_3(ValveObject:= ADR(ST03_422_Y64_6));(*Förderband Zuführung Stopper GST*)

(* Call ST03_422_Y64_7 Förderband links/rechts Züführung Stopper 1 AST/GST (Valve) *)
Analyze(InputExp:=  TRUE, DoAnalyze:= TRUE );
ST03_422_Y64_7.strAnlayse:=Analyze.OutString;
ST03_422_Y64_7(Enable  :=  Analyze.ExpResult,
                                sVisu:=Visu.ST03_422_Y64_7,
                                Reset:=gResetAll,
);
ST03_422_B64_2(ValveObject:= ADR(ST03_422_Y64_7));(*Förderband Zuführung Stopper Kamera AST*)
ST03_422_B64_1(ValveObject:= ADR(ST03_422_Y64_7));(*Förderband Zuführung Stopper Kamera GST*)


(* Call ST03_423_Y65_6 Förderband links/rechts Züführung Stopper 2 AST/GST (Valve) *)
Analyze(InputExp:=  TRUE, DoAnalyze:= TRUE );
ST03_423_Y65_6.strAnlayse:=Analyze.OutString;
ST03_423_Y65_6(Enable  :=  Analyze.ExpResult,
                                sVisu:=Visu.ST03_423_Y65_6,
                                Reset:=gResetAll,
);
ST03_423_B65_1(ValveObject:= ADR(ST03_423_Y65_6));(*Förderband Zuführung Stopper Kamera AST*)
ST03_423_B65_0(ValveObject:= ADR(ST03_423_Y65_6));(*Förderband Zuführung Stopper Kamera GST*)

(* Call ST03_423_Y65_7 Förderband links/rechts Züführung Stopper 3 AST/GST (Valve) *)
Analyze(InputExp:=  TRUE, DoAnalyze:= TRUE );
ST03_423_Y65_7.strAnlayse:=Analyze.OutString;
ST03_423_Y65_7(Enable  :=  Analyze.ExpResult,
                                sVisu:=Visu.ST03_423_Y65_7,
                                Reset:=gResetAll,
);
ST03_423_B65_3(ValveObject:= ADR(ST03_423_Y65_7));(*Förderband Zuführung Stopper Kamera AST*)
ST03_423_B65_4(ValveObject:= ADR(ST03_423_Y65_7));(*Förderband Zuführung Stopper Kamera GST*)

(* Call ST03_33F4 Steckdosenleise Tintenstrahldrucker  (DigIn) *)
ST03_33F4(		sVisu:=Visu.ST03_33F4,
				Reset:=gResetAll,
);
(* Call ST03_70U3_1 Bereit/ Im Druck Tintenstrahldrucker Frontseite   (DigIn) *)
ST03_70U3_1(sVisu:=Visu.ST03_70U3_1,
                                Reset:=gResetAll,
);
(* Call ST03_70U3_2 Tank voll Tintenstrahldrucker Frontseite   (DigIn) *)
ST03_70U3_2(	sVisu:=Visu.ST03_70U3_2,
				Reset:=gResetAll,
);
(* Call ST03_70U3_3 Fehler/Störung Tintenstrahldrucker Frontseite   (DigIn) *)
ST03_70U3_3(	sVisu:=Visu.ST03_70U3_3,
				Reset:=gResetAll,
);
(* Call ST03_71U3_1 Bereit/ Im Druck Tintenstrahldrucker Rückseite   (DigIn) *)
ST03_71U3_1(sVisu:=Visu.ST03_71U3_1,
                                Reset:=gResetAll,
);
(* Call ST03_71U3_2 Tank voll Tintenstrahldrucker Rückseite   (DigIn) *)
ST03_71U3_2(	sVisu:=Visu.ST03_71U3_2,
				Reset:=gResetAll,
);
(* Call ST03_71U3_3 Fehler/Störung Tintenstrahldrucker Rückseite   (DigIn) *)
ST03_71U3_3(	sVisu:=Visu.ST03_71U3_3,
				Reset:=gResetAll,
);
(* Call ST03_PLAN_70V1_1 Start  Bedrucken Tintenstrahldrucker Frontseite (DigOutIn) *)
ST03_PLAN_70V1_1(	sVisu:=Visu.ST03_PLAN_70V1_1,
						Reset:=gResetAll,
);
(* Call ST03_PLAN_70V1_1 Start  Bedrucken Tintenstrahldrucker Rückseite (DigOutIn) *)
ST03_PLAN_71V1_2(	sVisu:=Visu.ST03_PLAN_71V1_2,
						Reset:=gResetAll,
);
IF NOT MP.ST02.SensopartEthernet THEN
	(**Sensopart Kamera links*)
	ST03_8_80_A1(
		b_kamera_aktiv:=MP.ST03.FrontCamOn,
		st_Description:= 'Sensopart Kamera links',
		b_reset:=gResetAll );

	(**Sensopart Kamera rechts*)
	ST03_8_85_A1(
		b_kamera_aktiv:=MP.ST03.BackCamOn,
		st_Description:= 'Sensopart Kamera rechts',
		b_reset:=gResetAll );
ELSE
	(**Sensopart Kamera links*)
	IF MP.ST02.SensopartIPAdress <>''  THEN
		ST03_8_90_A1(
				Activated := MP.ST03.FrontCamOn,
				st_Description:= 'Sensopart Kamera links',
				);
		ST03_8_90_A1.s_IpAdress := MP.ST02.SensopartIPAdress;
		ST03_8_90_A1.i_CmdPort := 2006;
		ST03_8_90_A1.i_DataPort :=2005;
END_IF
	(**Sensopart Kamera rechts*)
	IF MP.ST02.SensopartIPAdress2 <>''  THEN
		ST03_8_95_A1(
				Activated := MP.ST03.BackCamOn,
				st_Description:= 'Sensopart Kamera rechts',
				);
		ST03_8_95_A1.s_IpAdress := MP.ST02.SensopartIPAdress2;
		ST03_8_95_A1.i_CmdPort := 2006;
		ST03_8_95_A1.i_DataPort :=2005;
	END_IF
END_IF

(* Init ST03_S18 ST02 Druckschalter Wartungseinheit Hauptluft Tintenstrahldrucker min.6 bar (DigIn)
nur bei 160 pol*)	
ST03_S18(	sVisu:=Visu.ST03_S18,
			Reset:=gResetAll,
);
(* Call ST03_H6 Signalsäule GR Bedruckung IO(DigOutIn) *)
ST03_H6(	sVisu:=Visu.ST03_H6,
			Reset:=gResetAll,
);
(* Call ST03_H7 Signalsäule RD Sammelstörung Bedruckung IO(DigOutIn) *)
ST03_H7(	sVisu:=Visu.ST03_H7,
			Reset:=gResetAll,
);
END_ACTION
ACTION call_7pol:
(* Call ST03_512_XG1 Zuführung  frei zum Ablegen ISK SP Maschine (DigIn) *)
ST03_512_XG1(sVisu:=Visu.ST03_512_XG1,
                                Reset:=gResetAll,
);
(* Call ST03_515_Y72_0 ISK Klemmer 1 AST/GST  (Valve) *)
Analyze(InputExp:=  TRUE, DoAnalyze:= TRUE );
ST03_515_Y72_0.strAnlayse:=Analyze.OutString;
ST03_515_Y72_0(Enable  :=  Analyze.ExpResult,
                                sVisu:=Visu.ST03_515_Y72_0,
                                Reset:=gResetAll,
);
ST03_512_B69_1(ValveObject:= ADR(ST03_515_Y72_0));(*ISK Klemmer 2 GST*)
ST03_512_B69_2(ValveObject:= ADR(ST03_515_Y72_0));(*ISK Klemmer 2 AST*)
ST03_512_B69_3(ValveObject:= ADR(ST03_515_Y72_0));(*ISK Klemmer 1 GST*)
ST03_512_B69_4(ValveObject:= ADR(ST03_515_Y72_0));(*ISK Klemmer 1 AST*)

(* Call ST03_515_Y72_1 Rinne schwenkern AST/GST  (Valve) *)
Analyze(InputExp:=  TRUE, DoAnalyze:= TRUE );
ST03_515_Y72_1.strAnlayse:=Analyze.OutString;
ST03_515_Y72_1(Enable  :=  Analyze.ExpResult,
                                sVisu:=Visu.ST03_515_Y72_1,
                                Reset:=gResetAll,
);
ST03_512_B69_5(ValveObject:= ADR(ST03_515_Y72_1));(*ISK Klemmer schwenkern 0° AST*)
ST03_512_B69_6(ValveObject:= ADR(ST03_515_Y72_1));(*ISK Klemmer schwenkern 180° GST*)

(* Call ST03_514_B71_7 Führungsschiene frei zum schwenken (DigIn) *)
ST03_514_B71_7(sVisu:=Visu.ST03_514_B71_7,
                                Reset:=gResetAll,
);
(* Call ST03_515_Y72_2 Führungsschiene  Zuführung Vereinzler AST/GST  (Valve) *)
Analyze(InputExp:=  TRUE, DoAnalyze:= TRUE );
ST03_515_Y72_2.strAnlayse:=Analyze.OutString;
ST03_515_Y72_2(Enable  :=  Analyze.ExpResult,
                                sVisu:=Visu.ST03_515_Y72_2,
                                Reset:=gResetAll,
);
ST03_513_B70_0(ValveObject:= ADR(ST03_515_Y72_2));(*Führungsschiene  Zuführung Vereinzler AST*)
ST03_513_B70_1(ValveObject:= ADR(ST03_515_Y72_2));(*Führungsschiene  Zuführung Vereinzler GST*)

(* Call ST03_515_Y72_3 Führungsschiene  Zuführung Stopper AST/GST  (Valve) *)
Analyze(InputExp:=  TRUE, DoAnalyze:= TRUE );
ST03_515_Y72_3.strAnlayse:=Analyze.OutString;
ST03_515_Y72_3(Enable  :=  Analyze.ExpResult,
                                sVisu:=Visu.ST03_515_Y72_3,
                                Reset:=gResetAll,
);
ST03_513_B70_2(ValveObject:= ADR(ST03_515_Y72_3));(*Führungsschiene  Zuführung Stopper AST*)
ST03_513_B70_3(ValveObject:= ADR(ST03_515_Y72_3));(*Führungsschiene  Zuführung Stopper GST*)

(* Call ST03_513_B70_4 ISK anwesend am Stopper(DigIn) *)
ST03_513_B70_4(sVisu:=Visu.ST03_513_B70_4,
                                Reset:=gResetAll,
);
(* Call ST03_515_Y72_4 Übergabeposition Stopper 1 AST/GST  (Valve) *)
Analyze(InputExp:=  TRUE, DoAnalyze:= TRUE );
ST03_515_Y72_4.strAnlayse:=Analyze.OutString;
ST03_515_Y72_4(Enable  :=  Analyze.ExpResult,
                                sVisu:=Visu.ST03_515_Y72_4,
                                Reset:=gResetAll,
);
ST03_513_B70_5(ValveObject:= ADR(ST03_515_Y72_4));(*Übergabeposition Stopper 1 AST*)
ST03_513_B70_6(ValveObject:= ADR(ST03_515_Y72_4));(*Übergabeposition Stopper 1 GST*)

(* Call ST03_513_B70_7 ISK auf Übergabeposition 1 (DigIn) *)
ST03_513_B70_7(sVisu:=Visu.ST03_513_B70_7,
                                Reset:=gResetAll,
);
(* Call ST03_515_Y72_5 Übergabeposition Stopper 2 AST/GST  (Valve) *)
Analyze(InputExp:=  TRUE, DoAnalyze:= TRUE );
ST03_515_Y72_5.strAnlayse:=Analyze.OutString;
ST03_515_Y72_5(Enable  :=  Analyze.ExpResult,
                                sVisu:=Visu.ST03_515_Y72_5,
                                Reset:=gResetAll,
);
ST03_514_B71_0(ValveObject:= ADR(ST03_515_Y72_5));(*Übergabeposition Stopper 2 AST*)
ST03_514_B71_1(ValveObject:= ADR(ST03_515_Y72_5));(*Übergabeposition Stopper 2 GST*)

(* Call ST03_514_B71_2 ISK auf Übergabeposition 2 (DigIn) *)
ST03_514_B71_2(sVisu:=Visu.ST03_514_B71_2,
                                Reset:=gResetAll,
);
(* Call ST03_515_Y72_6 Übergabeposition Stopper 3 AST/GST  (Valve) *)
Analyze(InputExp:=  TRUE, DoAnalyze:= TRUE );
ST03_515_Y72_6.strAnlayse:=Analyze.OutString;
ST03_515_Y72_6(Enable  :=  Analyze.ExpResult,
                                sVisu:=Visu.ST03_515_Y72_6,
                                Reset:=gResetAll,
);
ST03_514_B71_3(ValveObject:= ADR(ST03_515_Y72_6));(*Übergabeposition Stopper 3 AST*)
ST03_514_B71_4(ValveObject:= ADR(ST03_515_Y72_6));(*Übergabeposition Stopper 3 GST*)

(* Call ST03_514_B71_5 ISK auf Übergabeposition 3 (DigIn) *)
ST03_514_B71_5(sVisu:=Visu.ST03_514_B71_5,
                                Reset:=gResetAll,
);
(* Call ST03_514_B71_6 ISK auf Übergabeposition 4 (DigIn) *)
ST03_514_B71_6(sVisu:=Visu.ST03_514_B71_6,
                                Reset:=gResetAll,
);
END_ACTION
ACTION call_88pol:
(* Call ST03_501_B69_0 IZuführung  frei zum Ablegen ISK SP Maschine (DigIn) *)
ST03_501_B69_0(sVisu:=Visu.ST03_501_B69_0,
                                Reset:=gResetAll,
);
(* Call ST03_502_Y70_1 Förderband  Zuführung Vereinzler AST/GST  (Valve) *)
Analyze(InputExp:=  TRUE, DoAnalyze:= TRUE );
ST03_502_Y70_1.strAnlayse:=Analyze.OutString;
ST03_502_Y70_1(Enable  :=  Analyze.ExpResult,
                                sVisu:=Visu.ST03_502_Y70_1,
                                Reset:=gResetAll,
);
ST03_501_B69_1(ValveObject:= ADR(ST03_502_Y70_1));(*Förderband Zuführung Vereinzler   AST*)
ST03_501_B69_2(ValveObject:= ADR(ST03_502_Y70_1));(*Förderband Zuführung Vereinzler   GST*)

(* Call ST03_502_Y70_2 örderband  Züführung Stopper AST/GST  (Valve) *)
Analyze(InputExp:=  TRUE, DoAnalyze:= TRUE );
ST03_502_Y70_2.strAnlayse:=Analyze.OutString;
ST03_502_Y70_2(Enable  :=  Analyze.ExpResult,
                                sVisu:=Visu.ST03_502_Y70_2,
                                Reset:=gResetAll,
);
ST03_501_B69_3(ValveObject:= ADR(ST03_502_Y70_2));(*Förderband Zuführung Stopper   AST*)
ST03_501_B69_4(ValveObject:= ADR(ST03_502_Y70_2));(*Förderband Zuführung Stopper   GST*)

(* Call ST03_501_B69_5 SK anwesend am Vereinzler (DigIn) *)
ST03_501_B69_5(sVisu:=Visu.ST03_501_B69_5,
                                Reset:=gResetAll,
);
(* Call ST03_501_B69_6 SK anwesend am Stoper (DigIn) *)
ST03_501_B69_6(sVisu:=Visu.ST03_501_B69_6,
                                Reset:=gResetAll,
);
(* Call ST03_501_B69_7 ISK auf Abholposition Robi (DigIn) *)
ST03_501_B69_7(sVisu:=Visu.ST03_501_B69_7,
                                Reset:=gResetAll,
);
(* Call ST03_502_B70_0  ISK Lageerkennung (DigIn) *)
ST03_502_B70_0(sVisu:=Visu.ST03_502_B70_0,
                                Reset:=gResetAll,
);
END_ACTION
ACTION call_88polAMG:
(* Call ST03_521_B69_0 IZuführung  frei zum Ablegen ISK SP Maschine (DigIn) *)
ST03_521_B69_0(sVisu:=Visu.ST03_521_B69_0,
                                Reset:=gResetAll,
);
(* Call ST03_522_Y70_1  Zuführung Vereinzler AST/GST  (Valve) *)
Analyze(InputExp:=  TRUE, DoAnalyze:= TRUE );
ST03_522_Y70_1.strAnlayse:=Analyze.OutString;
ST03_522_Y70_1(Enable  :=  Analyze.ExpResult,
                                sVisu:=Visu.ST03_522_Y70_1,
                                Reset:=gResetAll,
);
ST03_521_B69_1(ValveObject:= ADR(ST03_522_Y70_1));(*  Zuführung Vereinzler eingefahren GST*)
ST03_521_B69_2(ValveObject:= ADR(ST03_522_Y70_1));(*  Zuführung Vereinzler ausgefahren AST*)

(* Call ST03_522_Y70_2  Züführung Stopper AST/GST  (Valve) *)
Analyze(InputExp:=  TRUE, DoAnalyze:= TRUE );
ST03_522_Y70_2.strAnlayse:=Analyze.OutString;
ST03_522_Y70_2(Enable  :=  Analyze.ExpResult,
                                sVisu:=Visu.ST03_522_Y70_2,
                                Reset:=gResetAll,
);
ST03_521_B69_3(ValveObject:= ADR(ST03_522_Y70_2));(* Zuführung Stopper  eingefahren  AST*)
ST03_521_B69_4(ValveObject:= ADR(ST03_522_Y70_2));(* Zuführung Stopper  ausgefahren GST*)


(* Call ST03_521_B69_6 SK anwesend am Stoper (DigIn) *)
ST03_521_B69_6(sVisu:=Visu.ST03_521_B69_6,
                                Reset:=gResetAll,
);
(* Call ST03_521_B69_7 ISK Lageerkennung links (DigIn) *)
ST03_521_B69_7(sVisu:=Visu.ST03_521_B69_7,
                                Reset:=gResetAll,
);
(* Call ST03_522_B70_0  ISK Lageerkennung rechts (DigIn) *)
ST03_522_B70_0(sVisu:=Visu.ST03_522_B70_0,
                                Reset:=gResetAll,
);
END_ACTION
ACTION call_92pol:
(* Call ST03_446_Y70_5 Förderband  Zuführung Vereinzler AST/GST  (Valve) *)
Analyze(InputExp:=  TRUE, DoAnalyze:= TRUE );
ST03_446_Y70_5.strAnlayse:=Analyze.OutString;
ST03_446_Y70_5(Enable  :=  Analyze.ExpResult,
                                sVisu:=Visu.ST03_446_Y70_5,
                                Reset:=gResetAll,
);
ST03_444_B69_0(ValveObject:= ADR(ST03_446_Y70_5));(*Förderband Zuführung Vereinzler   AST*)
ST03_444_B69_1(ValveObject:= ADR(ST03_446_Y70_5));(*Förderband Zuführung Vereinzler   GST*)

(* Call ST03_446_Y70_6 Förderband  Zuführung Stopper AST/GST  (Valve) *)
Analyze(InputExp:=  TRUE, DoAnalyze:= TRUE );
ST03_446_Y70_6.strAnlayse:=Analyze.OutString;
ST03_446_Y70_6(Enable  :=  Analyze.ExpResult,
                                sVisu:=Visu.ST03_446_Y70_6,
                                Reset:=gResetAll,
);
ST03_444_B69_2(ValveObject:= ADR(ST03_446_Y70_6));(*Förderband Zuführung Stopper   AST*)
ST03_444_B69_3(ValveObject:= ADR(ST03_446_Y70_6));(*Förderband Zuführung Stopper   GST*)

(* Call ST03_444_B69_4 Zuführung  frei zum Ablegen ISK SP Maschine Pos.1  (DigIn) *)
ST03_444_B69_4(sVisu:=Visu.ST03_444_B69_4,
                                Reset:=gResetAll,
);
(* Call ST03_444_B69_7 Zuführung  ISK anwesend am Stopper (DigIn) *)
ST03_444_B69_7(sVisu:=Visu.ST03_444_B69_7,
                                Reset:=gResetAll,
);
(* Call ST03_446_B70_4  ISK auf Übergabeposition zu Roboter  (DigIn) *)
ST03_446_B70_4(sVisu:=Visu.ST03_446_B70_4,
                                Reset:=gResetAll,
);
(* Call ST03_445_B70_1 Zuführung  ISK Lageerkennung links (DigIn) *)
ST03_445_B70_1(sVisu:=Visu.ST03_445_B70_1,
                                Reset:=gResetAll,
);
(* Call ST03_445_B70_2 Zuführung  ISK Lageerkennung links (DigIn) *)
ST03_445_B70_2(sVisu:=Visu.ST03_445_B70_2,
                                Reset:=gResetAll,
);
END_ACTION
ACTION call_NOX4pol:
ST03_8_100_A1(
		st_ctrl_in := ST03_8_100_A1.st_ctrl_in,
		Activated := MP.ST03.CamOn[1],
		st_Description:= 'Kamera Farberkennung',
		SensopartErgebnis:=TD.SensopartErgebnis,
		);
ST03_8_100_A1.s_IpAdress := MP.ST03.SensopartIPAdress[1];  		(* 'MP.SensopartIPAdress';*)
ST03_8_100_A1.i_CmdPort := 2006;
ST03_8_100_A1.i_DataPort :=2005;

(* Call ST03_492_Y70_0 Förderband  Zuführung Vereinzler AST/GST  (Valve) *)
Analyze(InputExp:=  TRUE, DoAnalyze:= TRUE );
ST03_492_Y70_0.strAnlayse:=Analyze.OutString;
ST03_492_Y70_0(Enable  :=  Analyze.ExpResult,
                                sVisu:=Visu.ST03_492_Y70_0,
                                Reset:=gResetAll,
);
ST03_491_B69_1(ValveObject:= ADR(ST03_492_Y70_0));(*Förderband Zuführung Vereinzler   AST*)
ST03_491_B69_2(ValveObject:= ADR(ST03_492_Y70_0));(*Förderband Zuführung Vereinzler   GST*)

(* Call ST03_492_Y70_1 Förderband  Zuführung Stopper AST/GST  (Valve) *)
Analyze(InputExp:=  TRUE, DoAnalyze:= TRUE );
ST03_492_Y70_1.strAnlayse:=Analyze.OutString;
ST03_492_Y70_1(Enable  :=  Analyze.ExpResult,
                                sVisu:=Visu.ST03_492_Y70_1,
                                Reset:=gResetAll,
);
ST03_491_B69_3(ValveObject:= ADR(ST03_492_Y70_1));(*Förderband Zuführung Stopper   AST*)
ST03_491_B69_4(ValveObject:= ADR(ST03_492_Y70_1));(*Förderband Zuführung Stopper   GST*)

(* Call ST03_491_B69_0 Zuführung  frei zum Ablegen ISK SP Maschine (DigIn) *)
ST03_491_B69_0(sVisu:=Visu.ST03_491_B69_0,
                                Reset:=gResetAll,
);
(* Call ST03_491_B69_5 SK anwesend am Stoper (DigIn) *)
ST03_491_B69_5(sVisu:=Visu.ST03_491_B69_5,
                                Reset:=gResetAll,
);
(* Call ST03_491_B69_7 ISK auf Abholposition Robi (DigIn) *)
ST03_491_B69_7(sVisu:=Visu.ST03_491_B69_7,
                                Reset:=gResetAll,
);
END_ACTION
ACTION call_NOX5_6pol:
(* Sensopart Kamera*)
ST03_8_100_A1(
		st_ctrl_in := ST03_8_100_A1.st_ctrl_in,
		st_Description:= 'Sensopart Kamera',
		st_InstName := 'ST03_8_100_A1',
		Activated := MP.ST03.CamOn[1],
		SensopartErgebnis:=TD.SensopartErgebnis,
		);
ST03_8_100_A1.s_IpAdress := MP.ST03.SensopartIPAdress[1];  		(* 'MP.SensopartIPAdress';*)
ST03_8_100_A1.i_CmdPort := 2006;
ST03_8_100_A1.i_DataPort :=2005;

(* Keyence Kamera*)
ST03_8_105_A1();

ST03_8_105_A1.sConfig.Description := 'Keyence Kamera';
ST03_8_105_A1.sConfig.InstName := 'ST03_8_105_A1';
ST03_8_105_A1.sConfig.Aktiv := MP.ST03.CamOn_KYE;


(* Call ST03_4x2_B69_0 Zuführung frei zum Ablegen ISK SP Maschine  (DigIn) *)
ST03_4x2_B69_0(sVisu:=Visu.ST03_4x2_B69_0,
                                Reset:=gResetAll,
);
(* Call ST03_4x2_B69_5 ISK anwesend am Stopper  (DigIn) *)
ST03_4x2_B69_5(sVisu:=Visu.ST03_4x2_B69_5,
                                Reset:=gResetAll,
);
(* Call ST03_4x3_B70_0 ISK anwesend Übergabeposition Stopper  (DigIn) *)
ST03_4x3_B70_0(sVisu:=Visu.ST03_4x3_B70_0,
                                Reset:=gResetAll,
);
(* Call ST03_4x3_B70_1 ISK anwesend Übergabeposition  (DigIn) *)
ST03_4x3_B70_1(sVisu:=Visu.ST03_4x3_B70_1,
                                Reset:=gResetAll,
);
(* Call ST03_4x3_Y70_5 Zuführung Vereinzler AST/GST  (Valve) *)
Analyze(InputExp:=  TRUE, DoAnalyze:= TRUE );
ST03_4x3_Y70_5.strAnlayse:=Analyze.OutString;
ST03_4x3_Y70_5(Enable  :=  Analyze.ExpResult,
                                sVisu:=Visu.ST03_4x3_Y70_5,
                                Reset:=gResetAll,
);
ST03_4x2_B69_1(ValveObject:= ADR(ST03_4x3_Y70_5));(*Zuführung Vereinzler GST eingefahren*)
ST03_4x2_B69_2(ValveObject:= ADR(ST03_4x3_Y70_5));(*Zuführung Vereinzler AST ausgefahren*)

(* Call ST03_4x3_Y70_6 Zuführung Stopper AST/GST  (Valve) *)
Analyze(InputExp:=  TRUE, DoAnalyze:= TRUE );
ST03_4x3_Y70_6.strAnlayse:=Analyze.OutString;
ST03_4x3_Y70_6(Enable  :=  Analyze.ExpResult,
                                sVisu:=Visu.ST03_4x3_Y70_6,
                                Reset:=gResetAll,
);
ST03_4x2_B69_3(ValveObject:= ADR(ST03_4x3_Y70_6));(*Zuführung Stopper AST eingefahren*)
ST03_4x2_B69_4(ValveObject:= ADR(ST03_4x3_Y70_6));(*Zuführung Stopper GST ausgefahren*)

(* Call ST03_4x3_Y70_7 Zuführung Stopper Übergabeposition AST/GST  (Valve) *)
Analyze(InputExp:=  TRUE, DoAnalyze:= TRUE );
ST03_4x3_Y70_7.strAnlayse:=Analyze.OutString;
ST03_4x3_Y70_7(Enable  :=  Analyze.ExpResult,
                                sVisu:=Visu.ST03_4x3_Y70_7,
                                Reset:=gResetAll,
);
ST03_4x2_B69_6(ValveObject:= ADR(ST03_4x3_Y70_7));(*Zuführung Stopper Übergabeposition AST eingefahren*)
ST03_4x2_B69_7(ValveObject:= ADR(ST03_4x3_Y70_7));(*Zuführung Stopper Übergabeposition GST ausgefahren*)
END_ACTION

(* POU Stations/ST_08_Palettierer/ST_08_CallFBs/ST08_CallFBs, ST *)
PROGRAM ST08_CallFBs


VAR


END_VAR
(*----------------------------------------------------------------------------------------------------------------------------------*)
(*Call ST08_180_M1 Abstapeln*)
ST08_180_M1.sConfig.Aktiv				:=MP.ST08.StapelMotor;
ST08_180_M1			(	sVisu:=Visu.ST08_180_M1,
						Override:= MP.ST08.Override_Abstapeln,
						Offset:=MP.ST08.PosOffsetAbstapeln.Pos,	(* in mm oder Grad am Antrieb*)
						Reset:=gResetAll,
						NotausOK := ST08_402_B51_4.BitInToCheck,
						sPosList:= TD.PosAbstapeln );
IF	ST08_180_M1.sVisuAxis.BtnTeach.Pressed THEN
	TD.PosAbstapeln[ST08_180_M1.sVisuAxis.PosNr].Pos:= STRING_TO_LREAL(LREAL_TO_FMTSTR(ST08_180_M1.sctrl.in.Position,2,TRUE));
END_IF
ST08_180_M1_ON	(
			b_Stop:= NOT ST08_402_B51_4.BitInToCheck ,
			Achse:=ST08_180_M1 );

(*Call ST08_185_M1 Aufstapeln*)
ST08_185_M1.sConfig.Aktiv				:=MP.ST08.StapelMotor;
ST08_185_M1			(	sVisu:=Visu.ST08_185_M1,
						Override:= MP.ST08.Override_Aufstapeln,
						Offset:=MP.ST08.PosOffsetAufstapeln.Pos,
						Reset:=gResetAll,
						NotausOK := ST08_402_B51_5.BitInToCheck,
						sPosList:= TD.PosAufstapeln);
IF	ST08_185_M1.sVisuAxis.BtnTeach.Pressed THEN
	TD.PosAufstapeln[ST08_185_M1.sVisuAxis.PosNr].Pos:= STRING_TO_LREAL(LREAL_TO_FMTSTR(ST08_185_M1.sctrl.in.Position,2,TRUE));
END_IF
ST08_185_M1_ON	(
			b_Stop:= NOT ST08_402_B51_5.BitInToCheck ,
			Achse:=ST08_185_M1 );

(*Call ST08_190_M1 Tray ausheben*)
ST08_190_M1.sConfig.Aktiv				:=MP.ST08.TrayAushebenMotor;
ST08_190_M1			(	sVisu:=Visu.ST08_190_M1,
						Override:= MP.ST08.Override_TrayAusheben,
						Offset:=MP.ST08.PosOffsetTrayAusheben.Pos,
						Reset:=gResetAll,
						NotausOK := ST00_350_B20_0.BitInToCheck,
						sPosList:= TD.PosTrayAusheben);
IF	ST08_190_M1.sVisuAxis.BtnTeach.Pressed THEN
	TD.PosAufstapeln[ST08_190_M1.sVisuAxis.PosNr].Pos:= STRING_TO_LREAL(LREAL_TO_FMTSTR(ST08_190_M1.sctrl.in.Position,2,TRUE));
END_IF
ST08_190_M1_ON	(
			b_Stop:= NOT ST00_350_B20_0.BitInToCheck ,
			Achse:=ST08_190_M1 );
(* ST08_190_M1 Tray ausheben --- Generating home position*)
IF MP.ST08.TrayAushebenMotor THEN
	gHomeOk:=gHomeOk AND ABS(ST08_190_M1.sPos.ist - TD.PosTrayAusheben[1].Pos) < 0.5; (*1=unten, 2=oben, *);
END_IF

(* Call ST08_400_B50_0 Traystapel vor Vereinzeler Einlaufband hinten (DigIn) *)
ST08_400_B50_0                 (sVisu:=Visu.ST08_400_B50_0,
                                Reset:=gResetAll,
);

(* Call ST08_401_B50_5 Traystapel vor Vereinzeler Einlaufband mitte (DigIn) *)
ST08_401_B50_5                 (sVisu:=Visu.ST08_401_B50_5,
                                Reset:=gResetAll,
);


(* Call ST08_402_B51_2  Traystapel vor Vereinzeler Einlaufband vorne (DigIn) *)
ST08_402_B51_2                 (sVisu:=Visu.ST08_402_B51_2,
                                Reset:=gResetAll,
);

(* Call ST08_402_B51_4 (* Luftzone 1 *) (DigIn) *)
ST08_402_B51_4                 (sVisu:=Visu.ST08_402_B51_4,
                                Reset:=gResetAll,
);
(* Call ST08_402_B51_5 (* Luftzone 2 *) (DigIn) *)
ST08_402_B51_5                 (sVisu:=Visu.ST08_402_B51_5,
                                Reset:=gResetAll,
);
(* Call ST08_404_B52_2 Traystapel in Ablageposition Isokörper (DigIn) *)
ST08_404_B52_2                 (sVisu:=Visu.ST08_404_B52_2,
                                Reset:=gResetAll,
);
(* Call ST08_404_B52_3 Traystapel richtig eingelegt Isokörper (DigIn) *)
ST08_404_B52_3                 (sVisu:=Visu.ST08_404_B52_3,
                                Reset:=gResetAll,
);

(* Call ST08_406_B54_3 Traystapel in Ausheber (DigIn) *)
ST08_406_B54_3                 (sVisu:=Visu.ST08_406_B54_3,
                                Reset:=gResetAll,
);
(* Call ST08_406_B54_0 Tray in Zwischenp. Entnahme Isokörper (Bandende) (DigIn) *)
ST08_406_B54_0                 (sVisu:=Visu.ST08_406_B54_0,
                                Reset:=gResetAll,
);

(* Call ST08_406_B54_6 Tray aus Entnahme ausgelaufen (Bandende) (DigIn) *)
ST08_406_B54_6                 (sVisu:=Visu.ST08_406_B54_6,
                                Reset:=gResetAll,
);

(* Call ST08_407_B55_4 Tray in Aufstapelposition eingelaufen STN8 (DigIn) *)
ST08_407_B55_4                 (sVisu:=Visu.ST08_407_B55_4,
                                Reset:=gResetAll,
);
(* Call ST08_409_B55_5 Auslaufrollenbahn voll STN8 (DigIn) *)
ST08_409_B55_5                 (sVisu:=Visu.ST08_409_B55_5,
                                Reset:=gResetAll,
);


(* Call ST08_412_B58_4 Rüstsatz Förderband frei zum Ablegen ISK von SP Maschine Position 1 (DigIn) *)
ST08_412_B58_4                 (sVisu:=Visu.ST08_412_B58_4,
                                Reset:=gResetAll,
);

(* Call ST08_412_B58_5 Rüstsatz Förderband frei zum Ablegen ISK von SP Maschine Position 2 (DigIn) *)
ST08_412_B58_5                 (sVisu:=Visu.ST08_412_B58_5,
                                Reset:=gResetAll,
);

(* Call ST08_412_B58_6 Rüstsatz Förderband frei zum Ablegen ISK von SP Maschine Position 3 (DigIn) *)
ST08_412_B58_6                 (sVisu:=Visu.ST08_412_B58_6,
                                Reset:=gResetAll,
);

(* Call ST08_412_B58_5_35pol Lageerkennung links (DigIn) *)
ST08_412_B58_5_35pol                 (sVisu:=Visu.ST08_412_B58_5_35pol,
                                Reset:=gResetAll,
);

(* Call ST08_412_B58_6_35pol Lageerkennung rechts (DigIn) *)
ST08_412_B58_6_35pol                 (sVisu:=Visu.ST08_412_B58_6_35pol,
                                Reset:=gResetAll,
);

(* Call ST08_412_B58_7 Rüstsatz Förderband  ISK anwesend zum Vereinzeln (DigIn) *)
ST08_412_B58_7                 (sVisu:=Visu.ST08_412_B58_7,
                                Reset:=gResetAll,
);

(* Call ST08_412_B59_0 Rüstsatz Förderband ISK auf Übergabeposition Roboter Verpackung (DigIn) *)
ST08_412_B59_0                 (sVisu:=Visu.ST08_412_B59_0,
                                Reset:=gResetAll,
);

(* Call ST08_169_K1 Bandantrieb 1 Auslauf leere Trays Ein (DigOutIn) *)
ST08_169_K1                    (sVisu:=Visu.ST08_169_K1,
                                Reset:=gResetAll,
);
(* Call ST08_169_K2 Bandantrieb 4 Auslauf leere Trays Ein (DigOutIn) *)
ST08_169_K2                    (sVisu:=Visu.ST08_169_K2,
                                Reset:=gResetAll,
);
(* Call ST08_170_K1 Bandantrieb 2 Hubquereinheit Trays Ein (DigOutIn) *)
ST08_170_K1                    (sVisu:=Visu.ST08_170_K1,
                                Reset:=gResetAll,
);
(* Call ST08_170_K2 Bandantrieb 3 Hubquereinheit Trays Ein (DigOutIn) *)
ST08_170_K2                    (sVisu:=Visu.ST08_170_K2,
                                Reset:=gResetAll,
);

IF MP.ST08.Trayzufuhr_Verlaengerung THEN
	(* Call ST08_400_Y50_0 Stopper Traystapel Einlaufb. hinten links + rechts AST (Valve) *)
	Analyze         (InputExp:=  TRUE,
	                 DoAnalyze:= TRUE );
	ST08_400_Y50_0.strAnlayse:=Analyze.OutString;
	ST08_400_Y50_0                 (Enable  :=  Analyze.ExpResult,
	                                sVisu:=Visu.ST08_400_Y50_0,
	                                Reset:=gResetAll,
	);
	ST08_400_B50_4(ValveObject:= ADR(ST08_400_Y50_0));(*ST08_400_B50_4 Stopper Traystapel Einlaufband hinten rechts GST*)
END_IF

(* Call ST08_400_Y50_2 Stopper Traystapel Einlaufb. mitte links + rechts AST (Valve) *)
Analyze         (InputExp:=  TRUE,
                 DoAnalyze:= TRUE );
ST08_400_Y50_2.strAnlayse:=Analyze.OutString;
ST08_400_Y50_2                 (Enable  :=  Analyze.ExpResult,
                                sVisu:=Visu.ST08_400_Y50_2,
                                Reset:=gResetAll,
);
ST08_401_B51_1(ValveObject:= ADR(ST08_400_Y50_2));(*ST08_400_B50_4 Stopper Traystapel Einlaufband mitte rechts GST*)

(* Call ST08_402_Y50_4 Stopper Traystapel Einlaufb. vorne links + rechts AST (Valve) *)
Analyze         (InputExp:=  TRUE,
                 DoAnalyze:= TRUE );
ST08_402_Y50_4.strAnlayse:=Analyze.OutString;
ST08_402_Y50_4                 (Enable  :=  Analyze.ExpResult,
                                sVisu:=Visu.ST08_402_Y50_4,
                                Reset:=gResetAll,
);
ST08_402_B51_6(ValveObject:= ADR(ST08_402_Y50_4));(*ST08_400_B50_4 Stopper Traystapel Einlaufband vorne rechts GST*)

(* Call ST08_403_Y50_6 Vakuum 1 Einlauf STN8 AST (Valve) *)
Analyze         (InputExp:=  TRUE,
                 DoAnalyze:= TRUE );
ST08_403_Y50_6.strAnlayse:=Analyze.OutString;
ST08_403_Y50_6                 (Enable  :=  Analyze.ExpResult,
                                sVisu:=Visu.ST08_403_Y50_6,
                                Reset:=gResetAll,
);

(* Call ST08_403_Y50_7 Vakuum 2 Einlauf STN8 AST (Valve) *)
Analyze         (InputExp:=  TRUE,
                 DoAnalyze:= TRUE );
ST08_403_Y50_7.strAnlayse:=Analyze.OutString;
ST08_403_Y50_7                 (Enable  :=  Analyze.ExpResult,
                                sVisu:=Visu.ST08_403_Y50_7,
                                Reset:=gResetAll,
);


(* Call ST08_405_Y51_0 Hubtüre 2 Einlauf Isokörper STN8 AST (Valve) *)
Analyze         (InputExp:=  TRUE,
                 DoAnalyze:= TRUE );
ST08_405_Y51_0.strAnlayse:=Analyze.OutString;
ST08_405_Y51_0                 (Enable  :=  Analyze.ExpResult,
                                sVisu:=Visu.ST08_405_Y51_0,
                                Reset:=gResetAll,
);

IF NOT MP.ST03.SGM_3621 THEN
	ST08_405_B53_6(ValveObject:= ADR(ST08_405_Y51_0));(*ST08_405_B53_6 Hubtüre 2 Einlauf STN8 AST*)
	ST08_405_B53_7(ValveObject:= ADR(ST08_405_Y51_0));(*ST08_405_B53_6 Hubtüre 2 Einlauf STN8 GST*)
ELSE
	ST08_405_B53_6(ValveObject:= ADR(ST08_405_Y51_0));(*ST08_405_B53_6 Hubtüre 2 Einlauf STN8 AST*)
END_IF

(* Call ST08_404_Y51_6 Stopper Traystapel Isokörper AST (Valve) *)
Analyze         (InputExp:=  TRUE,
                 DoAnalyze:= TRUE );
ST08_404_Y51_6.strAnlayse:=Analyze.OutString;
ST08_404_Y51_6                 (Enable  :=  Analyze.ExpResult,
                                sVisu:=Visu.ST08_404_Y51_6,
                                Reset:=gResetAll,
);
ST08_404_B52_4(ValveObject:= ADR(ST08_404_Y51_6));(*ST08_404_B52_4 Stopper Traystapel Isokörper AST*)
ST08_404_B52_5(ValveObject:= ADR(ST08_404_Y51_6));(*ST08_404_B52_5 Stopper Traystapel Isokörper GST*)

(* Call ST08_406_Y51_2 Hubtüre 3 STN8 AST (Valve) *)
Analyze         (InputExp:=  TRUE,
                 DoAnalyze:= TRUE );
ST08_406_Y51_2.strAnlayse:=Analyze.OutString;
ST08_406_Y51_2                 (Enable  :=  Analyze.ExpResult,
                                sVisu:=Visu.ST08_406_Y51_2,
                                Reset:=gResetAll,
);

IF NOT MP.ST03.SGM_3621 THEN
	ST08_407_B55_0(ValveObject:= ADR(ST08_406_Y51_2));(*ST08_407_B55_0 Hubtüre 3 Auslauf STN8 AST*)
	ST08_407_B55_1(ValveObject:= ADR(ST08_406_Y51_2));(*ST08_407_B55_0 Hubtüre 3 Auslauf STN8 GST*)
ELSE
	ST08_407_B55_0(ValveObject:= ADR(ST08_406_Y51_2));(*ST08_407_B55_0 Hubtüre 3 Auslauf STN8 AST*)
END_IF

(* Call ST08_407_Y51_4 Hubtüre 4 Auslauf STN8 AST (Valve) *)
Analyze         (InputExp:=  TRUE,
                 DoAnalyze:= TRUE );
ST08_407_Y51_4.strAnlayse:=Analyze.OutString;
ST08_407_Y51_4                 (Enable  :=  Analyze.ExpResult,
                                sVisu:=Visu.ST08_407_Y51_4,
                                Reset:=gResetAll,
);

IF NOT MP.ST03.SGM_3621 THEN
	ST08_407_B55_2(ValveObject:= ADR(ST08_407_Y51_4));(*ST08_407_B55_2 Hubtüre 4 Auslauf STN8 AST*)
	ST08_407_B55_3(ValveObject:= ADR(ST08_407_Y51_4));(*ST08_407_B55_2 Hubtüre 4 Auslauf STN8 GST*)
ELSE
	ST08_407_B55_2(ValveObject:= ADR(ST08_407_Y51_4));(*ST08_407_B55_2 Hubtüre 4 Auslauf STN8 AST*)
END_IF

(* Call ST08_406_Y52_3 Ausheber Trays Entnahmepos. Isok. STN8 GST (Valve) *)
Analyze         (InputExp:=  TRUE,
                 DoAnalyze:= TRUE );
ST08_406_Y52_3.strAnlayse:=Analyze.OutString;
ST08_406_Y52_3                 (Enable  :=  Analyze.ExpResult,
                                sVisu:=Visu.ST08_406_Y52_3,
                                Reset:=gResetAll,
);
ST08_406_B54_4(ValveObject:= ADR(ST08_406_Y52_3));(*ST08_406_B54_4 Ausheber Trays Entnahmepos. Isok. STN8 AST*)
ST08_406_B54_5(ValveObject:= ADR(ST08_406_Y52_3));(*ST08_406_B54_5 Ausheber Trays Entnahmepos. Isok. STN8 GST*)


IF NOT MP.ST03.SGM_3621 THEN
	(* Stopper links + rechts Traystapel Auslaufband einfahren (Valve) *)
	Analyze         (InputExp:=  TRUE,
	                 DoAnalyze:= TRUE );
	ST08_400_Y52_5.strAnlayse:=Analyze.OutString;
	ST08_400_Y52_5                 (Enable  :=  Analyze.ExpResult,
	                                sVisu:=Visu.ST08_400_Y52_5,
	                                Reset:=gResetAll,
	);

	ST08_400_B50_1(ValveObject:= ADR(ST08_400_Y52_5));(*ST08_400_B50_1 Stopper links + rechts Traystapel Auslaufband eingefahren*)
	ST08_400_B50_2(ValveObject:= ADR(ST08_400_Y52_5));(*ST08_400_B50_2 Stopper links + rechts Traystapel Auslaufband ausgefahren*)
	ST08_400_B50_3(ValveObject:= ADR(ST08_400_Y52_5));(*ST08_400_B50_3 Stopper links + rechts Traystapel Auslaufband eingefahren*)
	ST08_400_B50_6(ValveObject:= ADR(ST08_400_Y52_5));(*ST08_400_B50_6 Stopper links + rechts Traystapel Auslaufband ausgefahren*)
END_IF


IF MP.ST08.Traystapel_schieben THEN
	IF MP.ST08.Trayzufuhr_Verlaengerung THEN
		(* Call ST08_401_Y52_4 Traystapel schieben hinten ausfahren AST (Valve) *)
		Analyze         (InputExp:=  TRUE,
		                 DoAnalyze:= TRUE );
		ST08_401_Y52_4.strAnlayse:=Analyze.OutString;
		ST08_401_Y52_4                 (Enable  :=  Analyze.ExpResult,
		                                sVisu:=Visu.ST08_401_Y52_4,
		                                Reset:=gResetAll,
		);
		ST08_401_B50_7(ValveObject:= ADR(ST08_401_Y52_4));(*ST08_401_B50_7 Traystapel schieben hinten*)

		(* Call ST08_402_Y52_6 Traystapel schieben mitte ausfahren AST (Valve) *)
		Analyze         (InputExp:=  TRUE,
		                 DoAnalyze:= TRUE );
		ST08_402_Y52_6.strAnlayse:=Analyze.OutString;
		ST08_402_Y52_6                 (Enable  :=  Analyze.ExpResult,
		                                sVisu:=Visu.ST08_402_Y52_6,
		                                Reset:=gResetAll,
		);
		ST08_402_B51_3(ValveObject:= ADR(ST08_402_Y52_6));(*ST08_402_B51_3 Traystapel schieben mitte*)
	END_IF

	(* Call ST08_402_Y52_7 Traystapel schieben vorne ausfahren AST (Valve) *)
	Analyze         (InputExp:=  TRUE,
	                 DoAnalyze:= TRUE );
	ST08_402_Y52_7.strAnlayse:=Analyze.OutString;
	ST08_402_Y52_7                 (Enable  :=  Analyze.ExpResult,
	                                sVisu:=Visu.ST08_402_Y52_7,
	                                Reset:=gResetAll,
	);
	ST08_402_B51_7(ValveObject:= ADR(ST08_402_Y52_7));(*ST08_402_B51_7 Traystapel schieben vorne*)
END_IF


IF	NOT MP.ST08.StapelMotor THEN
	(* Call ST08_404_Y53_0 Abstapelzylinder 1 Isokörper AST (Valve) *)
	Analyze         (InputExp:=  TRUE,
	                 DoAnalyze:= TRUE );
	ST08_404_Y53_0.strAnlayse:=Analyze.OutString;
	ST08_404_Y53_0                 (Enable  :=  Analyze.ExpResult,
	                                sVisu:=Visu.ST08_404_Y53_0,
	                                Reset:=gResetAll,
	);
	ST08_404_B52_6(ValveObject:= ADR(ST08_404_Y53_0));(*ST08_404_B52_6 Abstapelzylinder 1 Isokörper AST*)
	ST08_404_B52_7(ValveObject:= ADR(ST08_404_Y53_0));(*ST08_404_B52_7 Abstapelzylinder 1 Isokörper GST*)

	
	(* Call ST08_404_Y53_2 Abstapelzylinder 2 Isokörper AST (Valve) *)
	Analyze         (InputExp:=  TRUE,
	                 DoAnalyze:= TRUE );
	ST08_404_Y53_2.strAnlayse:=Analyze.OutString;
	ST08_404_Y53_2                 (Enable  :=  Analyze.ExpResult,
	                                sVisu:=Visu.ST08_404_Y53_2,
	                                Reset:=gResetAll,
	);
	ST08_404_B53_0(ValveObject:= ADR(ST08_404_Y53_2));(*ST08_404_B53_0 Abstapelzylinder 2 Isokörper AST*)
	ST08_404_B53_1(ValveObject:= ADR(ST08_404_Y53_2));(*ST08_404_B53_1 Abstapelzylinder 2 Isokörper GST*)

	(* Call ST08_408_Y54_2 Abstapelzylinder 1 STN8 AST (Valve) *)
	Analyze         (InputExp:=  TRUE,
	                 DoAnalyze:= TRUE );
	ST08_408_Y54_2.strAnlayse:=Analyze.OutString;
	ST08_408_Y54_2                 (Enable  :=  Analyze.ExpResult,
	                                sVisu:=Visu.ST08_408_Y54_2,
	                                Reset:=gResetAll,
	);
	ST08_408_B56_4(ValveObject:= ADR(ST08_408_Y54_2));(*ST08_408_B56_4 Abstapelzylinder 1 STN8 AST*)
	ST08_408_B56_5(ValveObject:= ADR(ST08_408_Y54_2));(*ST08_408_B56_5 Abstapelzylinder 1 STN8 GST*)
	
	
	(* Call ST08_408_Y54_4 Abstapelzylinder 2 STN8 AST (Valve) *) 
	Analyze         (InputExp:=  TRUE,
	                 DoAnalyze:= TRUE );
	ST08_408_Y54_4.strAnlayse:=Analyze.OutString;
	ST08_408_Y54_4                 (Enable  :=  Analyze.ExpResult,
	                                sVisu:=Visu.ST08_408_Y54_4,
	                                Reset:=gResetAll,
	);
	ST08_408_B56_6(ValveObject:= ADR(ST08_408_Y54_4));(*ST08_408_B56_6 Abstapelzylinder 2 STN8 AST*)
	ST08_408_B56_7(ValveObject:= ADR(ST08_408_Y54_4));(*ST08_408_B56_7 Abstapelzylinder 2 STN8 GST*)
END_IF

(* Call ST08_405_Y53_4 Rückhaltezylinder li+re Traystapel Isokörper AST (Valve) *)
Analyze         (InputExp:=  TRUE,
                 DoAnalyze:= TRUE );
ST08_405_Y53_4.strAnlayse:=Analyze.OutString;
ST08_405_Y53_4                 (Enable  :=  Analyze.ExpResult,
                                sVisu:=Visu.ST08_405_Y53_4,
                                Reset:=gResetAll,
);
ST08_405_B53_2(ValveObject:= ADR(ST08_405_Y53_4));(*ST08_405_B53_2 Rückhaltezylinder links Traystapel Isokörper AST*)
ST08_405_B53_3(ValveObject:= ADR(ST08_405_Y53_4));(*ST08_405_B53_3 Rückhaltezylinder links Traystapel Isokörper GST*)
ST08_405_B53_4(ValveObject:= ADR(ST08_405_Y53_4));(*ST08_405_B53_4 Rückhaltezylinder links Traystapel Isokörper AST*)
ST08_405_B53_5(ValveObject:= ADR(ST08_405_Y53_4));(*ST08_405_B53_5 Rückhaltezylinder links Traystapel Isokörper GST*)



(* Call ST08_408_Y54_0 Rückhaltezylinder li.+re. Auslauf STN8 AST (Valve) *)
Analyze         (InputExp:=  TRUE,
                 DoAnalyze:= TRUE );
ST08_408_Y54_0.strAnlayse:=Analyze.OutString;
ST08_408_Y54_0                 (Enable  :=  Analyze.ExpResult,
                                sVisu:=Visu.ST08_408_Y54_0,
                                Reset:=gResetAll,
);
ST08_408_B56_0(ValveObject:= ADR(ST08_408_Y54_0));(*ST08_408_B56_0 Rückhaltezylinder links Traystapel Isokörper AST*)
ST08_408_B56_1(ValveObject:= ADR(ST08_408_Y54_0));(*ST08_408_B56_1 Rückhaltezylinder links Traystapel Isokörper GST*)
ST08_408_B56_2(ValveObject:= ADR(ST08_408_Y54_0));(*ST08_408_B56_2 Rückhaltezylinder links Traystapel Isokörper AST*)
ST08_408_B56_3(ValveObject:= ADR(ST08_408_Y54_0));(*ST08_408_B56_3 Rückhaltezylinder links Traystapel Isokörper GST*)


